LIN {X 0,Y 488.788,Z 369.847,A -85,B 0,C 180,E1 23776.764,E2 23776.764} C_VEL
LIN {X 0,Y 488.831,Z 369.841,A -85,B 0,C 180,E1 23773.364,E2 23773.364} C_VEL
LIN {X 0,Y 488.776,Z 369.84,A -85,B 0,C 180,E1 23769.895,E2 23769.895} C_VEL
LIN {X 0,Y 488.771,Z 369.837,A -85,B 0,C 180,E1 23766.342,E2 23766.342} C_VEL
LIN {X 0,Y 488.82,Z 369.843,A -85,B 0,C 180,E1 23762.931,E2 23762.931} C_VEL
LIN {X 0,Y 488.772,Z 369.849,A -85,B 0,C 180,E1 23759.531,E2 23759.531} C_VEL
LIN {X 0,Y 488.762,Z 369.849,A -85,B 0,C 180,E1 23756.012,E2 23756.012} C_VEL
LIN {X 0,Y 488.816,Z 369.838,A -85,B 0,C 180,E1 23752.596,E2 23752.596} C_VEL
LIN {X 0,Y 488.767,Z 369.845,A -85,B 0,C 180,E1 23749.152,E2 23749.152} C_VEL
LIN {X 0,Y 488.75,Z 369.847,A -85,B 0,C 180,E1 23745.669,E2 23745.669} C_VEL
LIN {X 0,Y 488.801,Z 369.846,A -85,B 0,C 180,E1 23742.255,E2 23742.255} C_VEL
LIN {X 0,Y 488.77,Z 369.853,A -85,B 0,C 180,E1 23738.772,E2 23738.772} C_VEL
LIN {X 0,Y 488.748,Z 369.822,A -85,B 0,C 180,E1 23735.262,E2 23735.262} C_VEL
LIN {X 0,Y 488.792,Z 369.844,A -85,B 0,C 180,E1 23731.802,E2 23731.802} C_VEL
LIN {X 0,Y 488.773,Z 369.83,A -85,B 0,C 180,E1 23728.535,E2 23728.535} C_VEL
LIN {X 0,Y 488.76,Z 369.829,A -85,B 0,C 180,E1 23725.055,E2 23725.055} C_VEL
LIN {X 0,Y 488.805,Z 369.844,A -85,B 0,C 180,E1 23721.55,E2 23721.55} C_VEL
LIN {X 0,Y 488.797,Z 369.846,A -85,B 0,C 180,E1 23718.117,E2 23718.117} C_VEL
LIN {X 0,Y 488.832,Z 370.155,A -85,B 0,C 180,E1 23717.192,E2 23717.192} C_VEL
LIN {X 0,Y 490.288,Z 373.622,A -85,B 0,C 180,E1 23716.717,E2 23716.717} C_VEL
LIN {X 0,Y 496.839,Z 386.984,A -85,B 0,C 180,E1 23715.06,E2 23715.06} C_VEL
LIN {X 0,Y 507.598,Z 410.407,A -85,B 0,C 180,E1 23712.424,E2 23712.424} C_VEL
LIN {X 0,Y 505.734,Z 452.561,A -85,B 0,C 180,E1 23709.796,E2 23709.796} C_VEL
LIN {X 0,Y 508.868,Z 476.154,A -85,B 0,C 180,E1 23709.124,E2 23709.124} C_VEL
LIN {X 0,Y 505.724,Z 690.25,A -85,B 0,C 180,E1 23705.753,E2 23705.753} C_VEL
LIN {X 0,Y 504.658,Z 761.758,A -85,B 0,C 180,E1 23704.625,E2 23704.625} C_VEL
LIN {X 0,Y 503.792,Z 783.614,A -85,B 0,C 180,E1 23704.081,E2 23704.081} C_VEL
LIN {X 0,Y 502.692,Z 805.814,A -85,B 0,C 180,E1 23703.323,E2 23703.323} C_VEL
LIN {X 0,Y 501.534,Z 826.289,A -85,B 0,C 180,E1 23702.427,E2 23702.427} C_VEL
LIN {X 0,Y 500.044,Z 845.014,A -85,B 0,C 180,E1 23701.373,E2 23701.373} C_VEL
LIN {X 0,Y 498.307,Z 865.526,A -85,B 0,C 180,E1 23699.972,E2 23699.972} C_VEL
LIN {X 0,Y 496.641,Z 883.778,A -85,B 0,C 180,E1 23698.496,E2 23698.496} C_VEL
LIN {X 0,Y 494.933,Z 901.869,A -85,B 0,C 180,E1 23696.758,E2 23696.758} C_VEL
LIN {X 0,Y 493.326,Z 918.685,A -85,B 0,C 180,E1 23694.867,E2 23694.867} C_VEL
LIN {X 0,Y 491.919,Z 934.189,A -85,B 0,C 180,E1 23692.842,E2 23692.842} C_VEL
LIN {X 0,Y 490.709,Z 948.64,A -85,B 0,C 180,E1 23690.639,E2 23690.639} C_VEL
LIN {X 0,Y 489.722,Z 961.46,A -85,B 0,C 180,E1 23688.324,E2 23688.324} C_VEL
LIN {X 0,Y 488.984,Z 972.816,A -85,B 0,C 180,E1 23685.901,E2 23685.901} C_VEL
LIN {X 0,Y 488.492,Z 982.262,A -85,B 0,C 180,E1 23683.493,E2 23683.493} C_VEL
LIN {X 0,Y 488.185,Z 989.884,A -85,B 0,C 180,E1 23681.099,E2 23681.099} C_VEL
LIN {X 0,Y 488.014,Z 996.146,A -85,B 0,C 180,E1 23678.601,E2 23678.601} C_VEL
LIN {X 0,Y 487.941,Z 1000.823,A -85,B 0,C 180,E1 23676.117,E2 23676.117} C_VEL
LIN {X 0,Y 487.912,Z 1003.79,A -85,B 0,C 180,E1 23673.639,E2 23673.639} C_VEL
LIN {X 0,Y 487.908,Z 1005.304,A -85,B 0,C 180,E1 23671.057,E2 23671.057} C_VEL
LIN {X 0,Y 487.907,Z 1005.259,A -85,B 0,C 180,E1 23668.709,E2 23668.709} C_VEL
LIN {X 0,Y 487.911,Z 1003.672,A -85,B 0,C 180,E1 23666.241,E2 23666.241} C_VEL
LIN {X 0,Y 487.944,Z 1000.634,A -85,B 0,C 180,E1 23663.766,E2 23663.766} C_VEL
LIN {X 0,Y 488.016,Z 995.893,A -85,B 0,C 180,E1 23661.281,E2 23661.281} C_VEL
LIN {X 0,Y 488.205,Z 989.179,A -85,B 0,C 180,E1 23658.663,E2 23658.663} C_VEL
LIN {X 0,Y 488.532,Z 981.433,A -85,B 0,C 180,E1 23656.268,E2 23656.268} C_VEL
LIN {X 0,Y 489.043,Z 971.79,A -85,B 0,C 180,E1 23653.858,E2 23653.858} C_VEL
LIN {X 0,Y 489.806,Z 960.195,A -85,B 0,C 180,E1 23651.433,E2 23651.433} C_VEL
LIN {X 0,Y 490.765,Z 947.879,A -85,B 0,C 180,E1 23649.24,E2 23649.24} C_VEL
LIN {X 0,Y 491.917,Z 934.195,A -85,B 0,C 180,E1 23647.159,E2 23647.159} C_VEL
LIN {X 0,Y 493.326,Z 918.693,A -85,B 0,C 180,E1 23645.133,E2 23645.133} C_VEL
LIN {X 0,Y 494.944,Z 901.728,A -85,B 0,C 180,E1 23643.228,E2 23643.228} C_VEL
LIN {X 0,Y 496.642,Z 883.789,A -85,B 0,C 180,E1 23641.505,E2 23641.505} C_VEL
LIN {X 0,Y 498.307,Z 865.542,A -85,B 0,C 180,E1 23640.029,E2 23640.029} C_VEL
LIN {X 0,Y 500.043,Z 845.02,A -85,B 0,C 180,E1 23638.627,E2 23638.627} C_VEL
LIN {X 0,Y 501.533,Z 826.306,A -85,B 0,C 180,E1 23637.573,E2 23637.573} C_VEL
LIN {X 0,Y 502.7,Z 805.692,A -85,B 0,C 180,E1 23636.671,E2 23636.671} C_VEL
LIN {X 0,Y 503.838,Z 782.562,A -85,B 0,C 180,E1 23635.889,E2 23635.889} C_VEL
LIN {X 0,Y 504.681,Z 760.801,A -85,B 0,C 180,E1 23635.356,E2 23635.356} C_VEL
LIN {X 0,Y 507.814,Z 542.394,A -85,B 0,C 180,E1 23631.935,E2 23631.935} C_VEL
LIN {X 0,Y 508.709,Z 473.556,A -85,B 0,C 180,E1 23630.818,E2 23630.818} C_VEL
LIN {X 0,Y 505.659,Z 451.562,A -85,B 0,C 180,E1 23630.164,E2 23630.164} C_VEL
LIN {X 0,Y 507.487,Z 410.144,A -85,B 0,C 180,E1 23627.548,E2 23627.548} C_VEL
LIN {X 0,Y 496.402,Z 386,A -85,B 0,C 180,E1 23624.827,E2 23624.827} C_VEL
LIN {X 0,Y 490.187,Z 373.48,A -85,B 0,C 180,E1 23623.263,E2 23623.263} C_VEL
LIN {X 0,Y 488.827,Z 370.128,A -85,B 0,C 180,E1 23622.809,E2 23622.809} C_VEL
LIN {X 0,Y 488.765,Z 369.836,A -85,B 0,C 180,E1 23621.35,E2 23621.35} C_VEL
LIN {X 0,Y 488.818,Z 369.85,A -85,B 0,C 180,E1 23618.001,E2 23618.001} C_VEL
LIN {X 0,Y 488.785,Z 369.834,A -85,B 0,C 180,E1 23614.484,E2 23614.484} C_VEL
LIN {X 0,Y 488.756,Z 369.825,A -85,B 0,C 180,E1 23611.012,E2 23611.012} C_VEL
LIN {X 0,Y 488.805,Z 369.85,A -85,B 0,C 180,E1 23607.667,E2 23607.667} C_VEL
LIN {X 0,Y 488.766,Z 369.816,A -85,B 0,C 180,E1 23604.279,E2 23604.279} C_VEL
LIN {X 0,Y 488.752,Z 369.852,A -85,B 0,C 180,E1 23600.804,E2 23600.804} C_VEL
LIN {X 0,Y 488.797,Z 369.851,A -85,B 0,C 180,E1 23597.376,E2 23597.376} C_VEL
LIN {X 0,Y 488.766,Z 369.847,A -85,B 0,C 180,E1 23593.968,E2 23593.968} C_VEL
LIN {X 0,Y 488.75,Z 369.847,A -85,B 0,C 180,E1 23590.49,E2 23590.49} C_VEL
LIN {X 0,Y 488.798,Z 369.839,A -85,B 0,C 180,E1 23587.05,E2 23587.05} C_VEL
LIN {X 0,Y 488.778,Z 369.848,A -85,B 0,C 180,E1 23583.636,E2 23583.636} C_VEL
LIN {X 0,Y 488.758,Z 369.85,A -85,B 0,C 180,E1 23580.117,E2 23580.117} C_VEL
LIN {X 0,Y 488.803,Z 369.848,A -85,B 0,C 180,E1 23576.716,E2 23576.716} C_VEL
LIN {X 0,Y 488.789,Z 369.837,A -85,B 0,C 180,E1 23573.304,E2 23573.304} C_VEL
LIN {X 0,Y 488.766,Z 369.839,A -85,B 0,C 180,E1 23569.867,E2 23569.867} C_VEL
LIN {X 0,Y 488.809,Z 369.841,A -85,B 0,C 180,E1 23566.394,E2 23566.394} C_VEL
LIN {X 0,Y 488.801,Z 369.849,A -85,B 0,C 180,E1 23562.991,E2 23562.991} C_VEL
LIN {X 0,Y 488.777,Z 369.846,A -85,B 0,C 180,E1 23559.521,E2 23559.521} C_VEL
LIN {X 0,Y 488.815,Z 369.843,A -85,B 0,C 180,E1 23556.096,E2 23556.096} C_VEL
LIN {X 0,Y 488.819,Z 369.838,A -85,B 0,C 180,E1 23552.577,E2 23552.577} C_VEL
LIN {X 0,Y 488.783,Z 369.839,A -85,B 0,C 180,E1 23549.106,E2 23549.106} C_VEL
LIN {X 0,Y 488.809,Z 369.841,A -85,B 0,C 180,E1 23545.628,E2 23545.628} C_VEL
LIN {X 0,Y 488.829,Z 369.815,A -85,B 0,C 180,E1 23542.134,E2 23542.134} C_VEL
LIN {X 0,Y 488.796,Z 369.848,A -85,B 0,C 180,E1 23538.645,E2 23538.645} C_VEL
LIN {X 0,Y 488.797,Z 369.824,A -85,B 0,C 180,E1 23535.047,E2 23535.047} C_VEL
LIN {X 0,Y 488.833,Z 369.816,A -85,B 0,C 180,E1 23531.501,E2 23531.501} C_VEL
LIN {X 0,Y 488.829,Z 369.836,A -85,B 0,C 180,E1 23527.858,E2 23527.858} C_VEL
LIN {X 0,Y 489.015,Z 370.806,A -85,B 0,C 180,E1 23527.599,E2 23527.599} C_VEL
LIN {X 0,Y 494.904,Z 385.117,A -85,B 0,C 180,E1 23525.426,E2 23525.426} C_VEL
LIN {X 0,Y 496.471,Z 389.129,A -85,B 0,C 180,E1 23525.033,E2 23525.033} C_VEL
LIN {X 0,Y 498.27,Z 395.004,A -85,B 0,C 180,E1 23524.736,E2 23524.736} C_VEL
LIN {X 0,Y 499.36,Z 402.645,A -85,B 0,C 180,E1 23524.515,E2 23524.515} C_VEL
LIN {X 0,Y 499.244,Z 418.921,A -85,B 0,C 180,E1 23524.239,E2 23524.239} C_VEL
LIN {X 0,Y 495.859,Z 645.556,A -85,B 0,C 180,E1 23520.716,E2 23520.716} C_VEL
LIN {X 0,Y 495.214,Z 666.185,A -85,B 0,C 180,E1 23520.218,E2 23520.218} C_VEL
LIN {X 0,Y 494.31,Z 684.909,A -85,B 0,C 180,E1 23519.567,E2 23519.567} C_VEL
LIN {X 0,Y 493.108,Z 703.249,A -85,B 0,C 180,E1 23518.718,E2 23518.718} C_VEL
LIN {X 0,Y 491.661,Z 720.942,A -85,B 0,C 180,E1 23517.686,E2 23517.686} C_VEL
LIN {X 0,Y 489.933,Z 739.495,A -85,B 0,C 180,E1 23516.355,E2 23516.355} C_VEL
LIN {X 0,Y 488.265,Z 755.721,A -85,B 0,C 180,E1 23514.948,E2 23514.948} C_VEL
LIN {X 0,Y 486.607,Z 771.11,A -85,B 0,C 180,E1 23513.361,E2 23513.361} C_VEL
LIN {X 0,Y 484.95,Z 785.984,A -85,B 0,C 180,E1 23511.528,E2 23511.528} C_VEL
LIN {X 0,Y 483.466,Z 799.353,A -85,B 0,C 180,E1 23509.572,E2 23509.572} C_VEL
LIN {X 0,Y 482.254,Z 811.31,A -85,B 0,C 180,E1 23507.493,E2 23507.493} C_VEL
LIN {X 0,Y 481.219,Z 822.432,A -85,B 0,C 180,E1 23505.175,E2 23505.175} C_VEL
LIN {X 0,Y 480.437,Z 834.341,A -85,B 0,C 180,E1 23502.132,E2 23502.132} C_VEL
LIN {X 0,Y 480.148,Z 841.698,A -85,B 0,C 180,E1 23499.83,E2 23499.83} C_VEL
LIN {X 0,Y 479.982,Z 847.651,A -85,B 0,C 180,E1 23497.419,E2 23497.419} C_VEL
LIN {X 0,Y 479.922,Z 851.89,A -85,B 0,C 180,E1 23495.019,E2 23495.019} C_VEL
LIN {X 0,Y 479.912,Z 854.507,A -85,B 0,C 180,E1 23492.626,E2 23492.626} C_VEL
LIN {X 0,Y 479.908,Z 855.453,A -85,B 0,C 180,E1 23490.238,E2 23490.238} C_VEL
LIN {X 0,Y 479.912,Z 854.828,A -85,B 0,C 180,E1 23487.851,E2 23487.851} C_VEL
LIN {X 0,Y 479.923,Z 852.487,A -85,B 0,C 180,E1 23485.34,E2 23485.34} C_VEL
LIN {X 0,Y 479.972,Z 848.604,A -85,B 0,C 180,E1 23482.94,E2 23482.94} C_VEL
LIN {X 0,Y 480.107,Z 842.998,A -85,B 0,C 180,E1 23480.531,E2 23480.531} C_VEL
LIN {X 0,Y 480.37,Z 835.903,A -85,B 0,C 180,E1 23478.231,E2 23478.231} C_VEL
LIN {X 0,Y 481.095,Z 824.054,A -85,B 0,C 180,E1 23475.108,E2 23475.108} C_VEL
LIN {X 0,Y 482.034,Z 813.717,A -85,B 0,C 180,E1 23472.871,E2 23472.871} C_VEL
LIN {X 0,Y 483.282,Z 801.241,A -85,B 0,C 180,E1 23470.634,E2 23470.634} C_VEL
LIN {X 0,Y 484.778,Z 787.534,A -85,B 0,C 180,E1 23468.59,E2 23468.59} C_VEL
LIN {X 0,Y 486.38,Z 772.874,A -85,B 0,C 180,E1 23466.755,E2 23466.755} C_VEL
LIN {X 0,Y 488.076,Z 757.496,A -85,B 0,C 180,E1 23465.136,E2 23465.136} C_VEL
LIN {X 0,Y 489.807,Z 740.762,A -85,B 0,C 180,E1 23463.656,E2 23463.656} C_VEL
LIN {X 0,Y 491.484,Z 723.176,A -85,B 0,C 180,E1 23462.368,E2 23462.368} C_VEL
LIN {X 0,Y 492.997,Z 704.892,A -85,B 0,C 180,E1 23461.274,E2 23461.274} C_VEL
LIN {X 0,Y 494.242,Z 686.026,A -85,B 0,C 180,E1 23460.391,E2 23460.391} C_VEL
LIN {X 0,Y 495.212,Z 666.341,A -85,B 0,C 180,E1 23459.696,E2 23459.696} C_VEL
LIN {X 0,Y 495.868,Z 645.599,A -85,B 0,C 180,E1 23459.193,E2 23459.193} C_VEL
LIN {X 0,Y 499.057,Z 431.182,A -85,B 0,C 180,E1 23455.86,E2 23455.86} C_VEL
LIN {X 0,Y 499.3,Z 407.126,A -85,B 0,C 180,E1 23455.472,E2 23455.472} C_VEL
LIN {X 0,Y 489.488,Z 390.831,A -85,B 0,C 180,E1 23454.288,E2 23454.288} C_VEL
LIN {X 0,Y 487.873,Z 387.972,A -85,B 0,C 180,E1 23454.05,E2 23454.05} C_VEL
LIN {X 0,Y 481.849,Z 373.753,A -85,B 0,C 180,E1 23451.855,E2 23451.855} C_VEL
LIN {X 0,Y 480.889,Z 371.018,A -85,B 0,C 180,E1 23451.375,E2 23451.375} C_VEL
LIN {X 0,Y 480.884,Z 370.81,A -85,B 0,C 180,E1 23447.926,E2 23447.926} C_VEL
LIN {X 0,Y 480.889,Z 370.803,A -85,B 0,C 180,E1 23444.316,E2 23444.316} C_VEL
LIN {X 0,Y 480.864,Z 370.834,A -85,B 0,C 180,E1 23440.761,E2 23440.761} C_VEL
LIN {X 0,Y 480.855,Z 370.824,A -85,B 0,C 180,E1 23437.086,E2 23437.086} C_VEL
LIN {X 0,Y 480.883,Z 370.829,A -85,B 0,C 180,E1 23433.521,E2 23433.521} C_VEL
LIN {X 0,Y 480.899,Z 370.824,A -85,B 0,C 180,E1 23429.897,E2 23429.897} C_VEL
LIN {X 0,Y 480.853,Z 370.829,A -85,B 0,C 180,E1 23426.348,E2 23426.348} C_VEL
LIN {X 0,Y 480.847,Z 370.83,A -85,B 0,C 180,E1 23422.754,E2 23422.754} C_VEL
LIN {X 0,Y 480.887,Z 370.824,A -85,B 0,C 180,E1 23419.289,E2 23419.289} C_VEL
LIN {X 0,Y 480.868,Z 370.833,A -85,B 0,C 180,E1 23415.716,E2 23415.716} C_VEL
LIN {X 0,Y 480.833,Z 370.837,A -85,B 0,C 180,E1 23412.246,E2 23412.246} C_VEL
LIN {X 0,Y 480.856,Z 370.839,A -85,B 0,C 180,E1 23408.731,E2 23408.731} C_VEL
LIN {X 0,Y 480.875,Z 370.824,A -85,B 0,C 180,E1 23405.249,E2 23405.249} C_VEL
LIN {X 0,Y 480.827,Z 370.827,A -85,B 0,C 180,E1 23401.788,E2 23401.788} C_VEL
LIN {X 0,Y 480.831,Z 370.832,A -85,B 0,C 180,E1 23398.213,E2 23398.213} C_VEL
LIN {X 0,Y 480.879,Z 370.837,A -85,B 0,C 180,E1 23394.751,E2 23394.751} C_VEL
LIN {X 0,Y 480.821,Z 370.837,A -85,B 0,C 180,E1 23391.389,E2 23391.389} C_VEL
LIN {X 0,Y 480.815,Z 370.839,A -85,B 0,C 180,E1 23387.754,E2 23387.754} C_VEL
LIN {X 0,Y 480.859,Z 370.831,A -85,B 0,C 180,E1 23384.288,E2 23384.288} C_VEL
LIN {X 0,Y 480.83,Z 370.831,A -85,B 0,C 180,E1 23380.819,E2 23380.819} C_VEL
LIN {X 0,Y 480.811,Z 370.828,A -85,B 0,C 180,E1 23377.374,E2 23377.374} C_VEL
LIN {X 0,Y 480.856,Z 370.825,A -85,B 0,C 180,E1 23373.921,E2 23373.921} C_VEL
LIN {X 0,Y 480.833,Z 370.816,A -85,B 0,C 180,E1 23370.598,E2 23370.598} C_VEL
LIN {X 0,Y 480.823,Z 370.842,A -85,B 0,C 180,E1 23367.13,E2 23367.13} C_VEL
LIN {X 0,Y 480.864,Z 370.809,A -85,B 0,C 180,E1 23363.659,E2 23363.659} C_VEL
LIN {X 0,Y 480.842,Z 370.812,A -85,B 0,C 180,E1 23360.291,E2 23360.291} C_VEL
LIN {X 0,Y 480.881,Z 370.964,A -85,B 0,C 180,E1 23358.051,E2 23358.051} C_VEL
LIN {X 0,Y 481.309,Z 372.589,A -85,B 0,C 180,E1 23357.777,E2 23357.777} C_VEL
LIN {X 0,Y 488.746,Z 387.377,A -85,B 0,C 180,E1 23355.847,E2 23355.847} C_VEL
LIN {X 0,Y 498.284,Z 408.17,A -85,B 0,C 180,E1 23353.416,E2 23353.416} C_VEL
LIN {X 0,Y 500.866,Z 414.181,A -85,B 0,C 180,E1 23352.763,E2 23352.763} C_VEL
LIN {X 0,Y 499.003,Z 451.774,A -85,B 0,C 180,E1 23350.384,E2 23350.384} C_VEL
LIN {X 0,Y 502.359,Z 477.415,A -85,B 0,C 180,E1 23349.638,E2 23349.638} C_VEL
LIN {X 0,Y 498.808,Z 694.303,A -85,B 0,C 180,E1 23346.163,E2 23346.163} C_VEL
LIN {X 0,Y 497.703,Z 760.723,A -85,B 0,C 180,E1 23345.096,E2 23345.096} C_VEL
LIN {X 0,Y 496.779,Z 782.356,A -85,B 0,C 180,E1 23344.552,E2 23344.552} C_VEL
LIN {X 0,Y 495.548,Z 804.985,A -85,B 0,C 180,E1 23343.77,E2 23343.77} C_VEL
LIN {X 0,Y 494.251,Z 826.148,A -85,B 0,C 180,E1 23342.827,E2 23342.827} C_VEL
LIN {X 0,Y 492.717,Z 846.558,A -85,B 0,C 180,E1 23341.704,E2 23341.704} C_VEL
LIN {X 0,Y 491.223,Z 865.433,A -85,B 0,C 180,E1 23340.45,E2 23340.45} C_VEL
LIN {X 0,Y 489.581,Z 882.526,A -85,B 0,C 180,E1 23339.063,E2 23339.063} C_VEL
LIN {X 0,Y 487.818,Z 899.472,A -85,B 0,C 180,E1 23337.44,E2 23337.44} C_VEL
LIN {X 0,Y 486.066,Z 916.658,A -85,B 0,C 180,E1 23335.526,E2 23335.526} C_VEL
LIN {X 0,Y 484.509,Z 932.49,A -85,B 0,C 180,E1 23333.469,E2 23333.469} C_VEL
LIN {X 0,Y 483.124,Z 947.102,A -85,B 0,C 180,E1 23331.232,E2 23331.232} C_VEL
LIN {X 0,Y 482.029,Z 959.88,A -85,B 0,C 180,E1 23328.939,E2 23328.939} C_VEL
LIN {X 0,Y 481.194,Z 971.27,A -85,B 0,C 180,E1 23326.538,E2 23326.538} C_VEL
LIN {X 0,Y 480.617,Z 980.974,A -85,B 0,C 180,E1 23324.086,E2 23324.086} C_VEL
LIN {X 0,Y 480.251,Z 988.824,A -85,B 0,C 180,E1 23321.65,E2 23321.65} C_VEL
LIN {X 0,Y 480.046,Z 995.384,A -85,B 0,C 180,E1 23319.107,E2 23319.107} C_VEL
LIN {X 0,Y 479.956,Z 1000.019,A -85,B 0,C 180,E1 23316.699,E2 23316.699} C_VEL
LIN {X 0,Y 479.915,Z 1003.446,A -85,B 0,C 180,E1 23314.062,E2 23314.062} C_VEL
LIN {X 0,Y 479.9,Z 1005.209,A -85,B 0,C 180,E1 23311.552,E2 23311.552} C_VEL
LIN {X 0,Y 479.903,Z 1005.326,A -85,B 0,C 180,E1 23309.045,E2 23309.045} C_VEL
LIN {X 0,Y 479.912,Z 1003.899,A -85,B 0,C 180,E1 23306.417,E2 23306.417} C_VEL
LIN {X 0,Y 479.943,Z 1000.98,A -85,B 0,C 180,E1 23303.902,E2 23303.902} C_VEL
LIN {X 0,Y 480.02,Z 996.401,A -85,B 0,C 180,E1 23301.376,E2 23301.376} C_VEL
LIN {X 0,Y 480.203,Z 990.238,A -85,B 0,C 180,E1 23298.836,E2 23298.836} C_VEL
LIN {X 0,Y 480.548,Z 982.419,A -85,B 0,C 180,E1 23296.328,E2 23296.328} C_VEL
LIN {X 0,Y 481.099,Z 972.817,A -85,B 0,C 180,E1 23293.832,E2 23293.832} C_VEL
LIN {X 0,Y 481.911,Z 961.463,A -85,B 0,C 180,E1 23291.369,E2 23291.369} C_VEL
LIN {X 0,Y 482.93,Z 949.363,A -85,B 0,C 180,E1 23289.141,E2 23289.141} C_VEL
LIN {X 0,Y 484.149,Z 935.883,A -85,B 0,C 180,E1 23287.028,E2 23287.028} C_VEL
LIN {X 0,Y 485.751,Z 919.705,A -85,B 0,C 180,E1 23284.849,E2 23284.849} C_VEL
LIN {X 0,Y 487.435,Z 903.548,A -85,B 0,C 180,E1 23282.98,E2 23282.98} C_VEL
LIN {X 0,Y 489.185,Z 886.121,A -85,B 0,C 180,E1 23281.263,E2 23281.263} C_VEL
LIN {X 0,Y 491,Z 867.941,A -85,B 0,C 180,E1 23279.739,E2 23279.739} C_VEL
LIN {X 0,Y 492.26,Z 852.622,A -85,B 0,C 180,E1 23278.673,E2 23278.673} C_VEL
LIN {X 0,Y 493.82,Z 831.791,A -85,B 0,C 180,E1 23277.465,E2 23277.465} C_VEL
LIN {X 0,Y 495.244,Z 810.72,A -85,B 0,C 180,E1 23276.461,E2 23276.461} C_VEL
LIN {X 0,Y 496.444,Z 788.83,A -85,B 0,C 180,E1 23275.645,E2 23275.645} C_VEL
LIN {X 0,Y 497.445,Z 767.04,A -85,B 0,C 180,E1 23275.048,E2 23275.048} C_VEL
LIN {X 0,Y 498.113,Z 742.947,A -85,B 0,C 180,E1 23274.597,E2 23274.597} C_VEL
LIN {X 0,Y 501.442,Z 527.679,A -85,B 0,C 180,E1 23271.181,E2 23271.181} C_VEL
LIN {X 0,Y 502.21,Z 474.909,A -85,B 0,C 180,E1 23270.305,E2 23270.305} C_VEL
LIN {X 0,Y 498.951,Z 450.509,A -85,B 0,C 180,E1 23269.558,E2 23269.558} C_VEL
LIN {X 0,Y 500.826,Z 413.756,A -85,B 0,C 180,E1 23267.204,E2 23267.204} C_VEL
LIN {X 0,Y 490.266,Z 390.634,A -85,B 0,C 180,E1 23264.552,E2 23264.552} C_VEL
LIN {X 0,Y 482.4,Z 374.624,A -85,B 0,C 180,E1 23262.507,E2 23262.507} C_VEL
LIN {X 0,Y 480.92,Z 371.178,A -85,B 0,C 180,E1 23262.025,E2 23262.025} C_VEL
LIN {X 0,Y 480.826,Z 370.823,A -85,B 0,C 180,E1 23261.357,E2 23261.357} C_VEL
LIN {X 0,Y 480.877,Z 370.839,A -85,B 0,C 180,E1 23257.985,E2 23257.985} C_VEL
LIN {X 0,Y 480.857,Z 370.822,A -85,B 0,C 180,E1 23254.371,E2 23254.371} C_VEL
LIN {X 0,Y 480.817,Z 370.81,A -85,B 0,C 180,E1 23250.906,E2 23250.906} C_VEL
LIN {X 0,Y 480.841,Z 370.84,A -85,B 0,C 180,E1 23247.401,E2 23247.401} C_VEL
LIN {X 0,Y 480.862,Z 370.799,A -85,B 0,C 180,E1 23243.92,E2 23243.92} C_VEL
LIN {X 0,Y 480.812,Z 370.841,A -85,B 0,C 180,E1 23240.575,E2 23240.575} C_VEL
LIN {X 0,Y 480.821,Z 370.84,A -85,B 0,C 180,E1 23236.97,E2 23236.97} C_VEL
LIN {X 0,Y 480.874,Z 370.837,A -85,B 0,C 180,E1 23233.466,E2 23233.466} C_VEL
LIN {X 0,Y 480.825,Z 370.836,A -85,B 0,C 180,E1 23229.938,E2 23229.938} C_VEL
LIN {X 0,Y 480.815,Z 370.835,A -85,B 0,C 180,E1 23226.447,E2 23226.447} C_VEL
LIN {X 0,Y 480.866,Z 370.826,A -85,B 0,C 180,E1 23222.979,E2 23222.979} C_VEL
LIN {X 0,Y 480.842,Z 370.838,A -85,B 0,C 180,E1 23219.523,E2 23219.523} C_VEL
LIN {X 0,Y 480.825,Z 370.837,A -85,B 0,C 180,E1 23216.065,E2 23216.065} C_VEL
LIN {X 0,Y 480.867,Z 370.835,A -85,B 0,C 180,E1 23212.593,E2 23212.593} C_VEL
LIN {X 0,Y 480.862,Z 370.825,A -85,B 0,C 180,E1 23209.093,E2 23209.093} C_VEL
LIN {X 0,Y 480.83,Z 370.831,A -85,B 0,C 180,E1 23205.673,E2 23205.673} C_VEL
LIN {X 0,Y 480.866,Z 370.831,A -85,B 0,C 180,E1 23202.202,E2 23202.202} C_VEL
LIN {X 0,Y 480.887,Z 370.836,A -85,B 0,C 180,E1 23198.651,E2 23198.651} C_VEL
LIN {X 0,Y 480.843,Z 370.836,A -85,B 0,C 180,E1 23195.163,E2 23195.163} C_VEL
LIN {X 0,Y 480.852,Z 370.835,A -85,B 0,C 180,E1 23191.564,E2 23191.564} C_VEL
LIN {X 0,Y 480.897,Z 370.833,A -85,B 0,C 180,E1 23188.122,E2 23188.122} C_VEL
LIN {X 0,Y 480.868,Z 370.836,A -85,B 0,C 180,E1 23184.541,E2 23184.541} C_VEL
LIN {X 0,Y 480.847,Z 370.801,A -85,B 0,C 180,E1 23180.946,E2 23180.946} C_VEL
LIN {X 0,Y 480.874,Z 370.828,A -85,B 0,C 180,E1 23177.39,E2 23177.39} C_VEL
LIN {X 0,Y 480.895,Z 370.83,A -85,B 0,C 180,E1 23173.811,E2 23173.811} C_VEL
LIN {X 0,Y 480.866,Z 370.813,A -85,B 0,C 180,E1 23170.262,E2 23170.262} C_VEL
LIN {X 0,Y 480.892,Z 371.07,A -85,B 0,C 180,E1 23168.509,E2 23168.509} C_VEL
LIN {X 0,Y 486.764,Z 385.17,A -85,B 0,C 180,E1 23166.264,E2 23166.264} C_VEL
LIN {X 0,Y 488.473,Z 389.111,A -85,B 0,C 180,E1 23165.747,E2 23165.747} C_VEL
LIN {X 0,Y 499.31,Z 407.175,A -85,B 0,C 180,E1 23164.434,E2 23164.434} C_VEL
LIN {X 0,Y 499.244,Z 418.921,A -85,B 0,C 180,E1 23164.239,E2 23164.239} C_VEL
LIN {X 0,Y 498.378,Z 426.618,A -85,B 0,C 180,E1 23164.185,E2 23164.185} C_VEL
LIN {X 0,Y 493.068,Z 447.174,A -85,B 0,C 180,E1 23164.308,E2 23164.308} C_VEL
LIN {X 0,Y 492.343,Z 453.787,A -85,B 0,C 180,E1 23164.26,E2 23164.26} C_VEL
LIN {X 0,Y 489.336,Z 650.297,A -85,B 0,C 180,E1 23161.184,E2 23161.184} C_VEL
LIN {X 0,Y 488.616,Z 670.204,A -85,B 0,C 180,E1 23160.663,E2 23160.663} C_VEL
LIN {X 0,Y 487.592,Z 689.333,A -85,B 0,C 180,E1 23159.951,E2 23159.951} C_VEL
LIN {X 0,Y 486.282,Z 707.632,A -85,B 0,C 180,E1 23159.066,E2 23159.066} C_VEL
LIN {X 0,Y 484.66,Z 726.308,A -85,B 0,C 180,E1 23157.921,E2 23157.921} C_VEL
LIN {X 0,Y 482.882,Z 743.342,A -85,B 0,C 180,E1 23156.63,E2 23156.63} C_VEL
LIN {X 0,Y 481.042,Z 759.594,A -85,B 0,C 180,E1 23155.151,E2 23155.151} C_VEL
LIN {X 0,Y 479.062,Z 776.072,A -85,B 0,C 180,E1 23153.36,E2 23153.36} C_VEL
LIN {X 0,Y 477.354,Z 790.398,A -85,B 0,C 180,E1 23151.5,E2 23151.5} C_VEL
LIN {X 0,Y 475.822,Z 803.326,A -85,B 0,C 180,E1 23149.516,E2 23149.516} C_VEL
LIN {X 0,Y 474.494,Z 815.492,A -85,B 0,C 180,E1 23147.282,E2 23147.282} C_VEL
LIN {X 0,Y 473.425,Z 826.079,A -85,B 0,C 180,E1 23144.929,E2 23144.929} C_VEL
LIN {X 0,Y 472.717,Z 834.698,A -85,B 0,C 180,E1 23142.582,E2 23142.582} C_VEL
LIN {X 0,Y 472.227,Z 842.036,A -85,B 0,C 180,E1 23140.081,E2 23140.081} C_VEL
LIN {X 0,Y 471.994,Z 847.767,A -85,B 0,C 180,E1 23137.519,E2 23137.519} C_VEL
LIN {X 0,Y 471.925,Z 852.209,A -85,B 0,C 180,E1 23134.861,E2 23134.861} C_VEL
LIN {X 0,Y 471.91,Z 854.643,A -85,B 0,C 180,E1 23132.428,E2 23132.428} C_VEL
LIN {X 0,Y 471.914,Z 855.497,A -85,B 0,C 180,E1 23130,E2 23130} C_VEL
LIN {X 0,Y 471.906,Z 854.691,A -85,B 0,C 180,E1 23127.571,E2 23127.571} C_VEL
LIN {X 0,Y 471.925,Z 852.325,A -85,B 0,C 180,E1 23125.139,E2 23125.139} C_VEL
LIN {X 0,Y 471.985,Z 848.136,A -85,B 0,C 180,E1 23122.576,E2 23122.576} C_VEL
LIN {X 0,Y 472.209,Z 842.497,A -85,B 0,C 180,E1 23120.002,E2 23120.002} C_VEL
LIN {X 0,Y 472.662,Z 835.424,A -85,B 0,C 180,E1 23117.54,E2 23117.54} C_VEL
LIN {X 0,Y 473.395,Z 826.454,A -85,B 0,C 180,E1 23115.069,E2 23115.069} C_VEL
LIN {X 0,Y 474.463,Z 815.719,A -85,B 0,C 180,E1 23112.675,E2 23112.675} C_VEL
LIN {X 0,Y 475.757,Z 803.827,A -85,B 0,C 180,E1 23110.48,E2 23110.48} C_VEL
LIN {X 0,Y 477.327,Z 790.636,A -85,B 0,C 180,E1 23108.443,E2 23108.443} C_VEL
LIN {X 0,Y 479.043,Z 776.263,A -85,B 0,C 180,E1 23106.573,E2 23106.573} C_VEL
LIN {X 0,Y 481.02,Z 759.818,A -85,B 0,C 180,E1 23104.781,E2 23104.781} C_VEL
LIN {X 0,Y 482.857,Z 743.605,A -85,B 0,C 180,E1 23103.301,E2 23103.301} C_VEL
LIN {X 0,Y 484.636,Z 726.593,A -85,B 0,C 180,E1 23102.008,E2 23102.008} C_VEL
LIN {X 0,Y 486.181,Z 708.756,A -85,B 0,C 180,E1 23100.907,E2 23100.907} C_VEL
LIN {X 0,Y 487.52,Z 690.499,A -85,B 0,C 180,E1 23100.009,E2 23100.009} C_VEL
LIN {X 0,Y 488.583,Z 671.076,A -85,B 0,C 180,E1 23099.274,E2 23099.274} C_VEL
LIN {X 0,Y 489.328,Z 651.025,A -85,B 0,C 180,E1 23098.74,E2 23098.74} C_VEL
LIN {X 0,Y 490.735,Z 559.481,A -85,B 0,C 180,E1 23097.289,E2 23097.289} C_VEL
LIN {X 0,Y 492.915,Z 410,A -85,B 0,C 180,E1 23094.944,E2 23094.944} C_VEL
LIN {X 0,Y 480.107,Z 389.093,A -85,B 0,C 180,E1 23093.327,E2 23093.327} C_VEL
LIN {X 0,Y 474.497,Z 375.687,A -85,B 0,C 180,E1 23091.23,E2 23091.23} C_VEL
LIN {X 0,Y 472.989,Z 372.055,A -85,B 0,C 180,E1 23090.581,E2 23090.581} C_VEL
LIN {X 0,Y 472.921,Z 371.817,A -85,B 0,C 180,E1 23087.192,E2 23087.192} C_VEL
LIN {X 0,Y 472.929,Z 371.796,A -85,B 0,C 180,E1 23083.523,E2 23083.523} C_VEL
LIN {X 0,Y 472.954,Z 371.794,A -85,B 0,C 180,E1 23079.885,E2 23079.885} C_VEL
LIN {X 0,Y 472.942,Z 371.82,A -85,B 0,C 180,E1 23076.296,E2 23076.296} C_VEL
LIN {X 0,Y 472.915,Z 371.825,A -85,B 0,C 180,E1 23072.713,E2 23072.713} C_VEL
LIN {X 0,Y 472.922,Z 371.827,A -85,B 0,C 180,E1 23069.096,E2 23069.096} C_VEL
LIN {X 0,Y 472.95,Z 371.821,A -85,B 0,C 180,E1 23065.494,E2 23065.494} C_VEL
LIN {X 0,Y 472.936,Z 371.818,A -85,B 0,C 180,E1 23061.871,E2 23061.871} C_VEL
LIN {X 0,Y 472.902,Z 371.82,A -85,B 0,C 180,E1 23058.335,E2 23058.335} C_VEL
LIN {X 0,Y 472.907,Z 371.817,A -85,B 0,C 180,E1 23054.698,E2 23054.698} C_VEL
LIN {X 0,Y 472.949,Z 371.815,A -85,B 0,C 180,E1 23051.216,E2 23051.216} C_VEL
LIN {X 0,Y 472.909,Z 371.825,A -85,B 0,C 180,E1 23047.655,E2 23047.655} C_VEL
LIN {X 0,Y 472.89,Z 371.827,A -85,B 0,C 180,E1 23044.123,E2 23044.123} C_VEL
LIN {X 0,Y 472.92,Z 371.821,A -85,B 0,C 180,E1 23040.606,E2 23040.606} C_VEL
LIN {X 0,Y 472.92,Z 371.815,A -85,B 0,C 180,E1 23037.092,E2 23037.092} C_VEL
LIN {X 0,Y 472.88,Z 371.823,A -85,B 0,C 180,E1 23033.566,E2 23033.566} C_VEL
LIN {X 0,Y 472.88,Z 371.825,A -85,B 0,C 180,E1 23029.893,E2 23029.893} C_VEL
LIN {X 0,Y 472.931,Z 371.825,A -85,B 0,C 180,E1 23026.428,E2 23026.428} C_VEL
LIN {X 0,Y 472.894,Z 371.829,A -85,B 0,C 180,E1 23022.861,E2 23022.861} C_VEL
LIN {X 0,Y 472.871,Z 371.831,A -85,B 0,C 180,E1 23019.323,E2 23019.323} C_VEL
LIN {X 0,Y 472.892,Z 371.789,A -85,B 0,C 180,E1 23015.784,E2 23015.784} C_VEL
LIN {X 0,Y 472.93,Z 371.827,A -85,B 0,C 180,E1 23012.282,E2 23012.282} C_VEL
LIN {X 0,Y 472.879,Z 371.799,A -85,B 0,C 180,E1 23008.899,E2 23008.899} C_VEL
LIN {X 0,Y 472.894,Z 371.805,A -85,B 0,C 180,E1 23005.326,E2 23005.326} C_VEL
LIN {X 0,Y 472.947,Z 371.822,A -85,B 0,C 180,E1 23001.726,E2 23001.726} C_VEL
LIN {X 0,Y 472.91,Z 371.967,A -85,B 0,C 180,E1 22998.888,E2 22998.888} C_VEL
LIN {X 0,Y 473.33,Z 373.614,A -85,B 0,C 180,E1 22998.611,E2 22998.611} C_VEL
LIN {X 0,Y 475.493,Z 377.652,A -85,B 0,C 180,E1 22998.035,E2 22998.035} C_VEL
LIN {X 0,Y 483.703,Z 394.372,A -85,B 0,C 180,E1 22995.845,E2 22995.845} C_VEL
LIN {X 0,Y 492.305,Z 413.289,A -85,B 0,C 180,E1 22993.611,E2 22993.611} C_VEL
LIN {X 0,Y 494.169,Z 417.443,A -85,B 0,C 180,E1 22993.143,E2 22993.143} C_VEL
LIN {X 0,Y 492.34,Z 451.126,A -85,B 0,C 180,E1 22990.983,E2 22990.983} C_VEL
LIN {X 0,Y 495.876,Z 478.8,A -85,B 0,C 180,E1 22990.161,E2 22990.161} C_VEL
LIN {X 0,Y 491.891,Z 700.139,A -85,B 0,C 180,E1 22986.556,E2 22986.556} C_VEL
LIN {X 0,Y 490.783,Z 759.683,A -85,B 0,C 180,E1 22985.58,E2 22985.58} C_VEL
LIN {X 0,Y 489.779,Z 781.518,A -85,B 0,C 180,E1 22985.023,E2 22985.023} C_VEL
LIN {X 0,Y 488.488,Z 803.557,A -85,B 0,C 180,E1 22984.252,E2 22984.252} C_VEL
LIN {X 0,Y 487.068,Z 824.691,A -85,B 0,C 180,E1 22983.304,E2 22983.304} C_VEL
LIN {X 0,Y 485.445,Z 845.141,A -85,B 0,C 180,E1 22982.165,E2 22982.165} C_VEL
LIN {X 0,Y 483.769,Z 865.033,A -85,B 0,C 180,E1 22980.832,E2 22980.832} C_VEL
LIN {X 0,Y 482.031,Z 884.412,A -85,B 0,C 180,E1 22979.307,E2 22979.307} C_VEL
LIN {X 0,Y 480.683,Z 898.049,A -85,B 0,C 180,E1 22978.038,E2 22978.038} C_VEL
LIN {X 0,Y 478.883,Z 914.63,A -85,B 0,C 180,E1 22976.203,E2 22976.203} C_VEL
LIN {X 0,Y 477.209,Z 929.734,A -85,B 0,C 180,E1 22974.244,E2 22974.244} C_VEL
LIN {X 0,Y 475.694,Z 944.376,A -85,B 0,C 180,E1 22972.039,E2 22972.039} C_VEL
LIN {X 0,Y 474.514,Z 957.008,A -85,B 0,C 180,E1 22969.829,E2 22969.829} C_VEL
LIN {X 0,Y 473.548,Z 968.537,A -85,B 0,C 180,E1 22967.445,E2 22967.445} C_VEL
LIN {X 0,Y 472.832,Z 978.68,A -85,B 0,C 180,E1 22964.949,E2 22964.949} C_VEL
LIN {X 0,Y 472.372,Z 987.056,A -85,B 0,C 180,E1 22962.468,E2 22962.468} C_VEL
LIN {X 0,Y 472.098,Z 993.687,A -85,B 0,C 180,E1 22959.996,E2 22959.996} C_VEL
LIN {X 0,Y 471.956,Z 998.987,A -85,B 0,C 180,E1 22957.425,E2 22957.425} C_VEL
LIN {X 0,Y 471.906,Z 1002.577,A -85,B 0,C 180,E1 22954.983,E2 22954.983} C_VEL
LIN {X 0,Y 471.901,Z 1004.746,A -85,B 0,C 180,E1 22952.429,E2 22952.429} C_VEL
LIN {X 0,Y 471.907,Z 1005.484,A -85,B 0,C 180,E1 22949.879,E2 22949.879} C_VEL
LIN {X 0,Y 471.897,Z 1004.677,A -85,B 0,C 180,E1 22947.45,E2 22947.45} C_VEL
LIN {X 0,Y 471.909,Z 1002.257,A -85,B 0,C 180,E1 22944.774,E2 22944.774} C_VEL
LIN {X 0,Y 471.969,Z 998.573,A -85,B 0,C 180,E1 22942.331,E2 22942.331} C_VEL
LIN {X 0,Y 472.125,Z 993.071,A -85,B 0,C 180,E1 22939.754,E2 22939.754} C_VEL
LIN {X 0,Y 472.415,Z 986.317,A -85,B 0,C 180,E1 22937.286,E2 22937.286} C_VEL
LIN {X 0,Y 472.896,Z 977.763,A -85,B 0,C 180,E1 22934.803,E2 22934.803} C_VEL
LIN {X 0,Y 473.633,Z 967.395,A -85,B 0,C 180,E1 22932.305,E2 22932.305} C_VEL
LIN {X 0,Y 474.635,Z 955.674,A -85,B 0,C 180,E1 22929.92,E2 22929.92} C_VEL
LIN {X 0,Y 475.896,Z 942.483,A -85,B 0,C 180,E1 22927.652,E2 22927.652} C_VEL
LIN {X 0,Y 477.404,Z 927.89,A -85,B 0,C 180,E1 22925.504,E2 22925.504} C_VEL
LIN {X 0,Y 479.165,Z 911.927,A -85,B 0,C 180,E1 22923.481,E2 22923.481} C_VEL
LIN {X 0,Y 480.897,Z 896.196,A -85,B 0,C 180,E1 22921.774,E2 22921.774} C_VEL
LIN {X 0,Y 482.577,Z 878.259,A -85,B 0,C 180,E1 22920.185,E2 22920.185} C_VEL
LIN {X 0,Y 484.317,Z 858.883,A -85,B 0,C 180,E1 22918.725,E2 22918.725} C_VEL
LIN {X 0,Y 485.983,Z 838.737,A -85,B 0,C 180,E1 22917.456,E2 22917.456} C_VEL
LIN {X 0,Y 487.521,Z 817.949,A -85,B 0,C 180,E1 22916.373,E2 22916.373} C_VEL
LIN {X 0,Y 488.968,Z 796.237,A -85,B 0,C 180,E1 22915.464,E2 22915.464} C_VEL
LIN {X 0,Y 490.115,Z 774.514,A -85,B 0,C 180,E1 22914.774,E2 22914.774} C_VEL
LIN {X 0,Y 491.008,Z 752.105,A -85,B 0,C 180,E1 22914.281,E2 22914.281} C_VEL
LIN {X 0,Y 494.724,Z 537.741,A -85,B 0,C 180,E1 22910.813,E2 22910.813} C_VEL
LIN {X 0,Y 495.726,Z 476.183,A -85,B 0,C 180,E1 22909.778,E2 22909.778} C_VEL
LIN {X 0,Y 492.285,Z 450.025,A -85,B 0,C 180,E1 22908.969,E2 22908.969} C_VEL
LIN {X 0,Y 494.168,Z 417.455,A -85,B 0,C 180,E1 22906.858,E2 22906.858} C_VEL
LIN {X 0,Y 484.143,Z 395.251,A -85,B 0,C 180,E1 22904.27,E2 22904.27} C_VEL
LIN {X 0,Y 476.245,Z 379.229,A -85,B 0,C 180,E1 22902.181,E2 22902.181} C_VEL
LIN {X 0,Y 474.648,Z 375.894,A -85,B 0,C 180,E1 22901.733,E2 22901.733} C_VEL
LIN {X 0,Y 472.964,Z 372.292,A -85,B 0,C 180,E1 22901.208,E2 22901.208} C_VEL
LIN {X 0,Y 472.902,Z 371.799,A -85,B 0,C 180,E1 22900.792,E2 22900.792} C_VEL
LIN {X 0,Y 472.886,Z 371.818,A -85,B 0,C 180,E1 22897.208,E2 22897.208} C_VEL
LIN {X 0,Y 472.911,Z 371.824,A -85,B 0,C 180,E1 22893.637,E2 22893.637} C_VEL
LIN {X 0,Y 472.934,Z 371.788,A -85,B 0,C 180,E1 22890.07,E2 22890.07} C_VEL
LIN {X 0,Y 472.881,Z 371.829,A -85,B 0,C 180,E1 22886.631,E2 22886.631} C_VEL
LIN {X 0,Y 472.875,Z 371.806,A -85,B 0,C 180,E1 22882.895,E2 22882.895} C_VEL
LIN {X 0,Y 472.921,Z 371.818,A -85,B 0,C 180,E1 22879.466,E2 22879.466} C_VEL
LIN {X 0,Y 472.893,Z 371.825,A -85,B 0,C 180,E1 22875.954,E2 22875.954} C_VEL
LIN {X 0,Y 472.87,Z 371.828,A -85,B 0,C 180,E1 22872.455,E2 22872.455} C_VEL
LIN {X 0,Y 472.896,Z 371.827,A -85,B 0,C 180,E1 22868.879,E2 22868.879} C_VEL
LIN {X 0,Y 472.92,Z 371.824,A -85,B 0,C 180,E1 22865.459,E2 22865.459} C_VEL
LIN {X 0,Y 472.882,Z 371.821,A -85,B 0,C 180,E1 22861.938,E2 22861.938} C_VEL
LIN {X 0,Y 472.887,Z 371.815,A -85,B 0,C 180,E1 22858.303,E2 22858.303} C_VEL
LIN {X 0,Y 472.937,Z 371.812,A -85,B 0,C 180,E1 22854.784,E2 22854.784} C_VEL
LIN {X 0,Y 472.903,Z 371.827,A -85,B 0,C 180,E1 22851.366,E2 22851.366} C_VEL
LIN {X 0,Y 472.892,Z 371.825,A -85,B 0,C 180,E1 22847.793,E2 22847.793} C_VEL
LIN {X 0,Y 472.929,Z 371.82,A -85,B 0,C 180,E1 22844.299,E2 22844.299} C_VEL
LIN {X 0,Y 472.939,Z 371.814,A -85,B 0,C 180,E1 22840.743,E2 22840.743} C_VEL
LIN {X 0,Y 472.903,Z 371.82,A -85,B 0,C 180,E1 22837.237,E2 22837.237} C_VEL
LIN {X 0,Y 472.905,Z 371.819,A -85,B 0,C 180,E1 22833.505,E2 22833.505} C_VEL
LIN {X 0,Y 472.96,Z 371.813,A -85,B 0,C 180,E1 22830.071,E2 22830.071} C_VEL
LIN {X 0,Y 472.935,Z 371.82,A -85,B 0,C 180,E1 22826.509,E2 22826.509} C_VEL
LIN {X 0,Y 472.91,Z 371.814,A -85,B 0,C 180,E1 22822.946,E2 22822.946} C_VEL
LIN {X 0,Y 472.932,Z 371.815,A -85,B 0,C 180,E1 22819.368,E2 22819.368} C_VEL
LIN {X 0,Y 472.951,Z 371.789,A -85,B 0,C 180,E1 22815.761,E2 22815.761} C_VEL
LIN {X 0,Y 472.931,Z 371.804,A -85,B 0,C 180,E1 22812.24,E2 22812.24} C_VEL
LIN {X 0,Y 472.99,Z 372.08,A -85,B 0,C 180,E1 22809.313,E2 22809.313} C_VEL
LIN {X 0,Y 475.816,Z 378.95,A -85,B 0,C 180,E1 22808.15,E2 22808.15} C_VEL
LIN {X 0,Y 480.422,Z 389.635,A -85,B 0,C 180,E1 22806.524,E2 22806.524} C_VEL
LIN {X 0,Y 493.039,Z 410.266,A -85,B 0,C 180,E1 22804.948,E2 22804.948} C_VEL
LIN {X 0,Y 492.343,Z 453.787,A -85,B 0,C 180,E1 22804.26,E2 22804.26} C_VEL
LIN {X 0,Y 491.412,Z 461.488,A -85,B 0,C 180,E1 22804.212,E2 22804.212} C_VEL
LIN {X 0,Y 486.12,Z 482.041,A -85,B 0,C 180,E1 22804.338,E2 22804.338} C_VEL
LIN {X 0,Y 485.42,Z 488.649,A -85,B 0,C 180,E1 22804.289,E2 22804.289} C_VEL
LIN {X 0,Y 482.841,Z 651.71,A -85,B 0,C 180,E1 22801.717,E2 22801.717} C_VEL
LIN {X 0,Y 482.104,Z 671.825,A -85,B 0,C 180,E1 22801.183,E2 22801.183} C_VEL
LIN {X 0,Y 481.06,Z 690.818,A -85,B 0,C 180,E1 22800.47,E2 22800.47} C_VEL
LIN {X 0,Y 479.738,Z 708.758,A -85,B 0,C 180,E1 22799.597,E2 22799.597} C_VEL
LIN {X 0,Y 478.078,Z 726.946,A -85,B 0,C 180,E1 22798.476,E2 22798.476} C_VEL
LIN {X 0,Y 476.194,Z 744.112,A -85,B 0,C 180,E1 22797.17,E2 22797.17} C_VEL
LIN {X 0,Y 474.217,Z 760.465,A -85,B 0,C 180,E1 22795.673,E2 22795.673} C_VEL
LIN {X 0,Y 472.149,Z 776.455,A -85,B 0,C 180,E1 22793.922,E2 22793.922} C_VEL
LIN {X 0,Y 470.258,Z 790.953,A -85,B 0,C 180,E1 22792.025,E2 22792.025} C_VEL
LIN {X 0,Y 468.53,Z 804.266,A -85,B 0,C 180,E1 22789.962,E2 22789.962} C_VEL
LIN {X 0,Y 467.052,Z 816.461,A -85,B 0,C 180,E1 22787.695,E2 22787.695} C_VEL
LIN {X 0,Y 465.848,Z 827.089,A -85,B 0,C 180,E1 22785.305,E2 22785.305} C_VEL
LIN {X 0,Y 465.041,Z 835.753,A -85,B 0,C 180,E1 22782.919,E2 22782.919} C_VEL
LIN {X 0,Y 464.465,Z 843.043,A -85,B 0,C 180,E1 22780.416,E2 22780.416} C_VEL
LIN {X 0,Y 464.166,Z 848.956,A -85,B 0,C 180,E1 22777.74,E2 22777.74} C_VEL
LIN {X 0,Y 464.003,Z 852.922,A -85,B 0,C 180,E1 22775.192,E2 22775.192} C_VEL
LIN {X 0,Y 463.954,Z 855.297,A -85,B 0,C 180,E1 22772.717,E2 22772.717} C_VEL
LIN {X 0,Y 463.944,Z 856.174,A -85,B 0,C 180,E1 22770.123,E2 22770.123} C_VEL
LIN {X 0,Y 463.945,Z 855.461,A -85,B 0,C 180,E1 22767.529,E2 22767.529} C_VEL
LIN {X 0,Y 464,Z 853.171,A -85,B 0,C 180,E1 22764.931,E2 22764.931} C_VEL
LIN {X 0,Y 464.154,Z 849.146,A -85,B 0,C 180,E1 22762.27,E2 22762.27} C_VEL
LIN {X 0,Y 464.441,Z 843.545,A -85,B 0,C 180,E1 22759.686,E2 22759.686} C_VEL
LIN {X 0,Y 464.982,Z 836.472,A -85,B 0,C 180,E1 22757.205,E2 22757.205} C_VEL
LIN {X 0,Y 465.817,Z 827.461,A -85,B 0,C 180,E1 22754.693,E2 22754.693} C_VEL
LIN {X 0,Y 466.997,Z 816.896,A -85,B 0,C 180,E1 22752.302,E2 22752.302} C_VEL
LIN {X 0,Y 468.462,Z 804.76,A -85,B 0,C 180,E1 22750.034,E2 22750.034} C_VEL
LIN {X 0,Y 470.132,Z 791.831,A -85,B 0,C 180,E1 22748.014,E2 22748.014} C_VEL
LIN {X 0,Y 471.987,Z 777.661,A -85,B 0,C 180,E1 22746.135,E2 22746.135} C_VEL
LIN {X 0,Y 474.046,Z 761.913,A -85,B 0,C 180,E1 22744.383,E2 22744.383} C_VEL
LIN {X 0,Y 476.003,Z 745.88,A -85,B 0,C 180,E1 22742.885,E2 22742.885} C_VEL
LIN {X 0,Y 477.869,Z 729.012,A -85,B 0,C 180,E1 22741.578,E2 22741.578} C_VEL
LIN {X 0,Y 479.508,Z 711.257,A -85,B 0,C 180,E1 22740.455,E2 22740.455} C_VEL
LIN {X 0,Y 480.987,Z 691.955,A -85,B 0,C 180,E1 22739.49,E2 22739.49} C_VEL
LIN {X 0,Y 482.072,Z 672.721,A -85,B 0,C 180,E1 22738.755,E2 22738.755} C_VEL
LIN {X 0,Y 482.835,Z 652.35,A -85,B 0,C 180,E1 22738.205,E2 22738.205} C_VEL
LIN {X 0,Y 484.255,Z 562.493,A -85,B 0,C 180,E1 22736.774,E2 22736.774} C_VEL
LIN {X 0,Y 486.599,Z 413.106,A -85,B 0,C 180,E1 22734.408,E2 22734.408} C_VEL
LIN {X 0,Y 474.04,Z 392.87,A -85,B 0,C 180,E1 22732.797,E2 22732.797} C_VEL
LIN {X 0,Y 472.03,Z 389.59,A -85,B 0,C 180,E1 22732.493,E2 22732.493} C_VEL
LIN {X 0,Y 466.178,Z 376.069,A -85,B 0,C 180,E1 22730.276,E2 22730.276} C_VEL
LIN {X 0,Y 465.029,Z 373.031,A -85,B 0,C 180,E1 22729.719,E2 22729.719} C_VEL
LIN {X 0,Y 465.014,Z 372.813,A -85,B 0,C 180,E1 22726.359,E2 22726.359} C_VEL
LIN {X 0,Y 464.994,Z 372.799,A -85,B 0,C 180,E1 22722.666,E2 22722.666} C_VEL
LIN {X 0,Y 464.975,Z 372.775,A -85,B 0,C 180,E1 22719.054,E2 22719.054} C_VEL
LIN {X 0,Y 464.997,Z 372.814,A -85,B 0,C 180,E1 22715.426,E2 22715.426} C_VEL
LIN {X 0,Y 465.018,Z 372.81,A -85,B 0,C 180,E1 22711.789,E2 22711.789} C_VEL
LIN {X 0,Y 464.992,Z 372.812,A -85,B 0,C 180,E1 22708.173,E2 22708.173} C_VEL
LIN {X 0,Y 464.968,Z 372.812,A -85,B 0,C 180,E1 22704.56,E2 22704.56} C_VEL
LIN {X 0,Y 464.977,Z 372.813,A -85,B 0,C 180,E1 22700.914,E2 22700.914} C_VEL
LIN {X 0,Y 465.013,Z 372.81,A -85,B 0,C 180,E1 22697.333,E2 22697.333} C_VEL
LIN {X 0,Y 464.977,Z 372.807,A -85,B 0,C 180,E1 22693.809,E2 22693.809} C_VEL
LIN {X 0,Y 464.955,Z 372.805,A -85,B 0,C 180,E1 22690.282,E2 22690.282} C_VEL
LIN {X 0,Y 464.987,Z 372.802,A -85,B 0,C 180,E1 22686.792,E2 22686.792} C_VEL
LIN {X 0,Y 464.993,Z 372.815,A -85,B 0,C 180,E1 22683.205,E2 22683.205} C_VEL
LIN {X 0,Y 464.948,Z 372.816,A -85,B 0,C 180,E1 22679.754,E2 22679.754} C_VEL
LIN {X 0,Y 464.949,Z 372.816,A -85,B 0,C 180,E1 22676.054,E2 22676.054} C_VEL
LIN {X 0,Y 464.997,Z 372.803,A -85,B 0,C 180,E1 22672.588,E2 22672.588} C_VEL
LIN {X 0,Y 464.962,Z 372.807,A -85,B 0,C 180,E1 22668.967,E2 22668.967} C_VEL
LIN {X 0,Y 464.932,Z 372.814,A -85,B 0,C 180,E1 22665.427,E2 22665.427} C_VEL
LIN {X 0,Y 464.944,Z 372.812,A -85,B 0,C 180,E1 22661.831,E2 22661.831} C_VEL
LIN {X 0,Y 464.997,Z 372.806,A -85,B 0,C 180,E1 22658.252,E2 22658.252} C_VEL
LIN {X 0,Y 464.954,Z 372.787,A -85,B 0,C 180,E1 22654.664,E2 22654.664} C_VEL
LIN {X 0,Y 464.94,Z 372.805,A -85,B 0,C 180,E1 22651.203,E2 22651.203} C_VEL
LIN {X 0,Y 464.977,Z 372.807,A -85,B 0,C 180,E1 22647.673,E2 22647.673} C_VEL
LIN {X 0,Y 464.989,Z 372.779,A -85,B 0,C 180,E1 22644.054,E2 22644.054} C_VEL
LIN {X 0,Y 464.948,Z 372.791,A -85,B 0,C 180,E1 22640.626,E2 22640.626} C_VEL
LIN {X 0,Y 465.053,Z 373.072,A -85,B 0,C 180,E1 22639.718,E2 22639.718} C_VEL
LIN {X 0,Y 466.509,Z 376.614,A -85,B 0,C 180,E1 22639.179,E2 22639.179} C_VEL
LIN {X 0,Y 472.003,Z 387.436,A -85,B 0,C 180,E1 22637.653,E2 22637.653} C_VEL
LIN {X 0,Y 480.238,Z 404.484,A -85,B 0,C 180,E1 22635.442,E2 22635.442} C_VEL
LIN {X 0,Y 487.461,Z 421.184,A -85,B 0,C 180,E1 22633.5,E2 22633.5} C_VEL
LIN {X 0,Y 485.741,Z 450.546,A -85,B 0,C 180,E1 22631.596,E2 22631.596} C_VEL
LIN {X 0,Y 489.43,Z 480.108,A -85,B 0,C 180,E1 22630.699,E2 22630.699} C_VEL
LIN {X 0,Y 485.115,Z 699.432,A -85,B 0,C 180,E1 22627.067,E2 22627.067} C_VEL
LIN {X 0,Y 483.878,Z 758.714,A -85,B 0,C 180,E1 22626.071,E2 22626.071} C_VEL
LIN {X 0,Y 482.778,Z 781.043,A -85,B 0,C 180,E1 22625.494,E2 22625.494} C_VEL
LIN {X 0,Y 481.424,Z 802.667,A -85,B 0,C 180,E1 22624.724,E2 22624.724} C_VEL
LIN {X 0,Y 479.877,Z 823.812,A -85,B 0,C 180,E1 22623.763,E2 22623.763} C_VEL
LIN {X 0,Y 478.104,Z 844.967,A -85,B 0,C 180,E1 22622.564,E2 22622.564} C_VEL
LIN {X 0,Y 476.325,Z 864.48,A -85,B 0,C 180,E1 22621.227,E2 22621.227} C_VEL
LIN {X 0,Y 474.49,Z 883.732,A -85,B 0,C 180,E1 22619.68,E2 22619.68} C_VEL
LIN {X 0,Y 472.579,Z 902.865,A -85,B 0,C 180,E1 22617.875,E2 22617.875} C_VEL
LIN {X 0,Y 471.029,Z 918.017,A -85,B 0,C 180,E1 22616.199,E2 22616.199} C_VEL
LIN {X 0,Y 469.674,Z 929.923,A -85,B 0,C 180,E1 22614.632,E2 22614.632} C_VEL
LIN {X 0,Y 468.009,Z 944.788,A -85,B 0,C 180,E1 22612.349,E2 22612.349} C_VEL
LIN {X 0,Y 466.701,Z 957.646,A -85,B 0,C 180,E1 22610.045,E2 22610.045} C_VEL
LIN {X 0,Y 465.65,Z 969.353,A -85,B 0,C 180,E1 22607.567,E2 22607.567} C_VEL
LIN {X 0,Y 464.892,Z 979.235,A -85,B 0,C 180,E1 22605.056,E2 22605.056} C_VEL
LIN {X 0,Y 464.382,Z 987.764,A -85,B 0,C 180,E1 22602.433,E2 22602.433} C_VEL
LIN {X 0,Y 464.1,Z 994.281,A -85,B 0,C 180,E1 22599.924,E2 22599.924} C_VEL
LIN {X 0,Y 463.959,Z 999.193,A -85,B 0,C 180,E1 22597.429,E2 22597.429} C_VEL
LIN {X 0,Y 463.907,Z 1002.736,A -85,B 0,C 180,E1 22594.946,E2 22594.946} C_VEL
LIN {X 0,Y 463.904,Z 1004.814,A -85,B 0,C 180,E1 22592.347,E2 22592.347} C_VEL
LIN {X 0,Y 463.9,Z 1005.462,A -85,B 0,C 180,E1 22589.753,E2 22589.753} C_VEL
LIN {X 0,Y 463.895,Z 1004.609,A -85,B 0,C 180,E1 22587.283,E2 22587.283} C_VEL
LIN {X 0,Y 463.918,Z 1002.097,A -85,B 0,C 180,E1 22584.559,E2 22584.559} C_VEL
LIN {X 0,Y 463.995,Z 998.366,A -85,B 0,C 180,E1 22582.074,E2 22582.074} C_VEL
LIN {X 0,Y 464.171,Z 992.768,A -85,B 0,C 180,E1 22579.451,E2 22579.451} C_VEL
LIN {X 0,Y 464.513,Z 985.506,A -85,B 0,C 180,E1 22576.813,E2 22576.813} C_VEL
LIN {X 0,Y 465.067,Z 976.843,A -85,B 0,C 180,E1 22574.285,E2 22574.285} C_VEL
LIN {X 0,Y 465.854,Z 966.82,A -85,B 0,C 180,E1 22571.87,E2 22571.87} C_VEL
LIN {X 0,Y 466.965,Z 954.972,A -85,B 0,C 180,E1 22569.445,E2 22569.445} C_VEL
LIN {X 0,Y 468.365,Z 941.711,A -85,B 0,C 180,E1 22567.14,E2 22567.14} C_VEL
LIN {X 0,Y 470.022,Z 926.963,A -85,B 0,C 180,E1 22564.959,E2 22564.959} C_VEL
LIN {X 0,Y 471.421,Z 914.439,A -85,B 0,C 180,E1 22563.373,E2 22563.373} C_VEL
LIN {X 0,Y 473.191,Z 896.749,A -85,B 0,C 180,E1 22561.523,E2 22561.523} C_VEL
LIN {X 0,Y 475.154,Z 876.638,A -85,B 0,C 180,E1 22559.721,E2 22559.721} C_VEL
LIN {X 0,Y 476.993,Z 857.447,A -85,B 0,C 180,E1 22558.259,E2 22558.259} C_VEL
LIN {X 0,Y 478.767,Z 837.296,A -85,B 0,C 180,E1 22556.975,E2 22556.975} C_VEL
LIN {X 0,Y 480.482,Z 815.954,A -85,B 0,C 180,E1 22555.856,E2 22555.856} C_VEL
LIN {X 0,Y 481.986,Z 794.117,A -85,B 0,C 180,E1 22554.943,E2 22554.943} C_VEL
LIN {X 0,Y 483.273,Z 771.824,A -85,B 0,C 180,E1 22554.239,E2 22554.239} C_VEL
LIN {X 0,Y 484.168,Z 749.63,A -85,B 0,C 180,E1 22553.76,E2 22553.76} C_VEL
LIN {X 0,Y 488.322,Z 532.592,A -85,B 0,C 180,E1 22550.18,E2 22550.18} C_VEL
LIN {X 0,Y 489.306,Z 477.576,A -85,B 0,C 180,E1 22549.241,E2 22549.241} C_VEL
LIN {X 0,Y 485.674,Z 449.43,A -85,B 0,C 180,E1 22548.357,E2 22548.357} C_VEL
LIN {X 0,Y 487.436,Z 420.909,A -85,B 0,C 180,E1 22546.478,E2 22546.478} C_VEL
LIN {X 0,Y 478.03,Z 399.862,A -85,B 0,C 180,E1 22543.981,E2 22543.981} C_VEL
LIN {X 0,Y 469.055,Z 381.378,A -85,B 0,C 180,E1 22541.524,E2 22541.524} C_VEL
LIN {X 0,Y 465.142,Z 373.591,A -85,B 0,C 180,E1 22540.398,E2 22540.398} C_VEL
LIN {X 0,Y 465.015,Z 372.823,A -85,B 0,C 180,E1 22540.169,E2 22540.169} C_VEL
LIN {X 0,Y 464.968,Z 372.788,A -85,B 0,C 180,E1 22536.559,E2 22536.559} C_VEL
LIN {X 0,Y 464.946,Z 372.82,A -85,B 0,C 180,E1 22532.961,E2 22532.961} C_VEL
LIN {X 0,Y 464.954,Z 372.788,A -85,B 0,C 180,E1 22529.36,E2 22529.36} C_VEL
LIN {X 0,Y 464.992,Z 372.792,A -85,B 0,C 180,E1 22525.881,E2 22525.881} C_VEL
LIN {X 0,Y 464.943,Z 372.805,A -85,B 0,C 180,E1 22522.373,E2 22522.373} C_VEL
LIN {X 0,Y 464.935,Z 372.81,A -85,B 0,C 180,E1 22518.819,E2 22518.819} C_VEL
LIN {X 0,Y 464.978,Z 372.805,A -85,B 0,C 180,E1 22515.336,E2 22515.336} C_VEL
LIN {X 0,Y 464.96,Z 372.81,A -85,B 0,C 180,E1 22511.788,E2 22511.788} C_VEL
LIN {X 0,Y 464.934,Z 372.816,A -85,B 0,C 180,E1 22508.284,E2 22508.284} C_VEL
LIN {X 0,Y 464.956,Z 372.816,A -85,B 0,C 180,E1 22504.687,E2 22504.687} C_VEL
LIN {X 0,Y 465.004,Z 372.812,A -85,B 0,C 180,E1 22501.109,E2 22501.109} C_VEL
LIN {X 0,Y 464.96,Z 372.805,A -85,B 0,C 180,E1 22497.535,E2 22497.535} C_VEL
LIN {X 0,Y 464.946,Z 372.802,A -85,B 0,C 180,E1 22493.951,E2 22493.951} C_VEL
LIN {X 0,Y 464.983,Z 372.804,A -85,B 0,C 180,E1 22490.469,E2 22490.469} C_VEL
LIN {X 0,Y 465.006,Z 372.811,A -85,B 0,C 180,E1 22486.825,E2 22486.825} C_VEL
LIN {X 0,Y 464.96,Z 372.815,A -85,B 0,C 180,E1 22483.381,E2 22483.381} C_VEL
LIN {X 0,Y 464.962,Z 372.813,A -85,B 0,C 180,E1 22479.632,E2 22479.632} C_VEL
LIN {X 0,Y 465.001,Z 372.806,A -85,B 0,C 180,E1 22476.156,E2 22476.156} C_VEL
LIN {X 0,Y 465.009,Z 372.803,A -85,B 0,C 180,E1 22472.465,E2 22472.465} C_VEL
LIN {X 0,Y 464.971,Z 372.805,A -85,B 0,C 180,E1 22468.929,E2 22468.929} C_VEL
LIN {X 0,Y 464.971,Z 372.811,A -85,B 0,C 180,E1 22465.22,E2 22465.22} C_VEL
LIN {X 0,Y 465.005,Z 372.772,A -85,B 0,C 180,E1 22461.697,E2 22461.697} C_VEL
LIN {X 0,Y 465.014,Z 372.81,A -85,B 0,C 180,E1 22458.033,E2 22458.033} C_VEL
LIN {X 0,Y 464.983,Z 372.794,A -85,B 0,C 180,E1 22454.446,E2 22454.446} C_VEL
LIN {X 0,Y 464.979,Z 372.783,A -85,B 0,C 180,E1 22450.806,E2 22450.806} C_VEL
LIN {X 0,Y 465.045,Z 373.127,A -85,B 0,C 180,E1 22450.152,E2 22450.152} C_VEL
LIN {X 0,Y 471.663,Z 388.704,A -85,B 0,C 180,E1 22447.549,E2 22447.549} C_VEL
LIN {X 0,Y 472.946,Z 391.163,A -85,B 0,C 180,E1 22447.254,E2 22447.254} C_VEL
LIN {X 0,Y 486.102,Z 412.269,A -85,B 0,C 180,E1 22445.56,E2 22445.56} C_VEL
LIN {X 0,Y 486.728,Z 413.817,A -85,B 0,C 180,E1 22445.473,E2 22445.473} C_VEL
LIN {X 0,Y 485.42,Z 488.649,A -85,B 0,C 180,E1 22444.289,E2 22444.289} C_VEL
LIN {X 0,Y 484.498,Z 496.351,A -85,B 0,C 180,E1 22444.24,E2 22444.24} C_VEL
LIN {X 0,Y 479.17,Z 516.895,A -85,B 0,C 180,E1 22444.375,E2 22444.375} C_VEL
LIN {X 0,Y 478.48,Z 523.503,A -85,B 0,C 180,E1 22444.324,E2 22444.324} C_VEL
LIN {X 0,Y 476.338,Z 653.019,A -85,B 0,C 180,E1 22442.257,E2 22442.257} C_VEL
LIN {X 0,Y 475.573,Z 673.191,A -85,B 0,C 180,E1 22441.714,E2 22441.714} C_VEL
LIN {X 0,Y 474.459,Z 692.562,A -85,B 0,C 180,E1 22440.975,E2 22440.975} C_VEL
LIN {X 0,Y 473.025,Z 711,A -85,B 0,C 180,E1 22440.06,E2 22440.06} C_VEL
LIN {X 0,Y 471.314,Z 729.186,A -85,B 0,C 180,E1 22438.923,E2 22438.923} C_VEL
LIN {X 0,Y 469.353,Z 746.307,A -85,B 0,C 180,E1 22437.6,E2 22437.6} C_VEL
LIN {X 0,Y 467.271,Z 762.565,A -85,B 0,C 180,E1 22436.083,E2 22436.083} C_VEL
LIN {X 0,Y 464.994,Z 778.934,A -85,B 0,C 180,E1 22434.246,E2 22434.246} C_VEL
LIN {X 0,Y 462.991,Z 793.139,A -85,B 0,C 180,E1 22432.336,E2 22432.336} C_VEL
LIN {X 0,Y 461.169,Z 805.974,A -85,B 0,C 180,E1 22430.295,E2 22430.295} C_VEL
LIN {X 0,Y 459.556,Z 818.067,A -85,B 0,C 180,E1 22427.994,E2 22427.994} C_VEL
LIN {X 0,Y 458.237,Z 828.623,A -85,B 0,C 180,E1 22425.566,E2 22425.566} C_VEL
LIN {X 0,Y 457.338,Z 837.226,A -85,B 0,C 180,E1 22423.141,E2 22423.141} C_VEL
LIN {X 0,Y 456.681,Z 844.545,A -85,B 0,C 180,E1 22420.566,E2 22420.566} C_VEL
LIN {X 0,Y 456.341,Z 850.235,A -85,B 0,C 180,E1 22417.933,E2 22417.933} C_VEL
LIN {X 0,Y 456.136,Z 854.276,A -85,B 0,C 180,E1 22415.281,E2 22415.281} C_VEL
LIN {X 0,Y 456.07,Z 856.631,A -85,B 0,C 180,E1 22412.764,E2 22412.764} C_VEL
LIN {X 0,Y 456.055,Z 857.502,A -85,B 0,C 180,E1 22410.125,E2 22410.125} C_VEL
LIN {X 0,Y 456.06,Z 856.795,A -85,B 0,C 180,E1 22407.487,E2 22407.487} C_VEL
LIN {X 0,Y 456.132,Z 854.526,A -85,B 0,C 180,E1 22404.844,E2 22404.844} C_VEL
LIN {X 0,Y 456.317,Z 850.63,A -85,B 0,C 180,E1 22402.193,E2 22402.193} C_VEL
LIN {X 0,Y 456.635,Z 845.336,A -85,B 0,C 180,E1 22399.657,E2 22399.657} C_VEL
LIN {X 0,Y 457.237,Z 838.358,A -85,B 0,C 180,E1 22397.113,E2 22397.113} C_VEL
LIN {X 0,Y 458.145,Z 829.482,A -85,B 0,C 180,E1 22394.56,E2 22394.56} C_VEL
LIN {X 0,Y 459.411,Z 819.057,A -85,B 0,C 180,E1 22392.131,E2 22392.131} C_VEL
LIN {X 0,Y 460.892,Z 807.795,A -85,B 0,C 180,E1 22389.943,E2 22389.943} C_VEL
LIN {X 0,Y 462.777,Z 794.557,A -85,B 0,C 180,E1 22387.786,E2 22387.786} C_VEL
LIN {X 0,Y 464.901,Z 779.615,A -85,B 0,C 180,E1 22385.748,E2 22385.748} C_VEL
LIN {X 0,Y 467.096,Z 764.008,A -85,B 0,C 180,E1 22383.974,E2 22383.974} C_VEL
LIN {X 0,Y 469.179,Z 747.892,A -85,B 0,C 180,E1 22382.441,E2 22382.441} C_VEL
LIN {X 0,Y 471.187,Z 730.305,A -85,B 0,C 180,E1 22381.068,E2 22381.068} C_VEL
LIN {X 0,Y 472.895,Z 712.404,A -85,B 0,C 180,E1 22379.93,E2 22379.93} C_VEL
LIN {X 0,Y 474.436,Z 692.957,A -85,B 0,C 180,E1 22378.952,E2 22378.952} C_VEL
LIN {X 0,Y 475.559,Z 673.611,A -85,B 0,C 180,E1 22378.209,E2 22378.209} C_VEL
LIN {X 0,Y 476.339,Z 653.272,A -85,B 0,C 180,E1 22377.657,E2 22377.657} C_VEL
LIN {X 0,Y 478.062,Z 549.408,A -85,B 0,C 180,E1 22375.993,E2 22375.993} C_VEL
LIN {X 0,Y 480.362,Z 416.278,A -85,B 0,C 180,E1 22373.863,E2 22373.863} C_VEL
LIN {X 0,Y 467.323,Z 395.375,A -85,B 0,C 180,E1 22372.138,E2 22372.138} C_VEL
LIN {X 0,Y 464.101,Z 390.277,A -85,B 0,C 180,E1 22371.647,E2 22371.647} C_VEL
LIN {X 0,Y 458.488,Z 377.46,A -85,B 0,C 180,E1 22369.473,E2 22369.473} C_VEL
LIN {X 0,Y 457.09,Z 373.984,A -85,B 0,C 180,E1 22368.806,E2 22368.806} C_VEL
LIN {X 0,Y 457.042,Z 373.775,A -85,B 0,C 180,E1 22365.138,E2 22365.138} C_VEL
LIN {X 0,Y 457.049,Z 373.805,A -85,B 0,C 180,E1 22361.384,E2 22361.384} C_VEL
LIN {X 0,Y 457.071,Z 373.764,A -85,B 0,C 180,E1 22357.772,E2 22357.772} C_VEL
LIN {X 0,Y 457.07,Z 373.792,A -85,B 0,C 180,E1 22354.057,E2 22354.057} C_VEL
LIN {X 0,Y 457.04,Z 373.791,A -85,B 0,C 180,E1 22350.473,E2 22350.473} C_VEL
LIN {X 0,Y 457.031,Z 373.794,A -85,B 0,C 180,E1 22346.787,E2 22346.787} C_VEL
LIN {X 0,Y 457.055,Z 373.79,A -85,B 0,C 180,E1 22343.19,E2 22343.19} C_VEL
LIN {X 0,Y 457.072,Z 373.789,A -85,B 0,C 180,E1 22339.554,E2 22339.554} C_VEL
LIN {X 0,Y 457.033,Z 373.801,A -85,B 0,C 180,E1 22336.001,E2 22336.001} C_VEL
LIN {X 0,Y 457.02,Z 373.804,A -85,B 0,C 180,E1 22332.381,E2 22332.381} C_VEL
LIN {X 0,Y 457.046,Z 373.804,A -85,B 0,C 180,E1 22328.809,E2 22328.809} C_VEL
LIN {X 0,Y 457.056,Z 373.789,A -85,B 0,C 180,E1 22325.272,E2 22325.272} C_VEL
LIN {X 0,Y 457.017,Z 373.791,A -85,B 0,C 180,E1 22321.63,E2 22321.63} C_VEL
LIN {X 0,Y 457.006,Z 373.798,A -85,B 0,C 180,E1 22317.994,E2 22317.994} C_VEL
LIN {X 0,Y 457.037,Z 373.802,A -85,B 0,C 180,E1 22314.448,E2 22314.448} C_VEL
LIN {X 0,Y 457.036,Z 373.804,A -85,B 0,C 180,E1 22310.938,E2 22310.938} C_VEL
LIN {X 0,Y 457,Z 373.805,A -85,B 0,C 180,E1 22307.343,E2 22307.343} C_VEL
LIN {X 0,Y 456.994,Z 373.808,A -85,B 0,C 180,E1 22303.606,E2 22303.606} C_VEL
LIN {X 0,Y 457.029,Z 373.803,A -85,B 0,C 180,E1 22300.045,E2 22300.045} C_VEL
LIN {X 0,Y 457.028,Z 373.765,A -85,B 0,C 180,E1 22296.537,E2 22296.537} C_VEL
LIN {X 0,Y 457.003,Z 373.809,A -85,B 0,C 180,E1 22292.931,E2 22292.931} C_VEL
LIN {X 0,Y 457.001,Z 373.77,A -85,B 0,C 180,E1 22289.206,E2 22289.206} C_VEL
LIN {X 0,Y 457.041,Z 373.782,A -85,B 0,C 180,E1 22285.638,E2 22285.638} C_VEL
LIN {X 0,Y 457.067,Z 373.803,A -85,B 0,C 180,E1 22281.911,E2 22281.911} C_VEL
LIN {X 0,Y 457.028,Z 373.926,A -85,B 0,C 180,E1 22280.711,E2 22280.711} C_VEL
LIN {X 0,Y 457.414,Z 375.457,A -85,B 0,C 180,E1 22280.418,E2 22280.418} C_VEL
LIN {X 0,Y 459.704,Z 379.692,A -85,B 0,C 180,E1 22279.761,E2 22279.761} C_VEL
LIN {X 0,Y 467.691,Z 395.438,A -85,B 0,C 180,E1 22277.502,E2 22277.502} C_VEL
LIN {X 0,Y 476.966,Z 415.567,A -85,B 0,C 180,E1 22274.942,E2 22274.942} C_VEL
LIN {X 0,Y 480.79,Z 424.483,A -85,B 0,C 180,E1 22273.897,E2 22273.897} C_VEL
LIN {X 0,Y 479.186,Z 449.852,A -85,B 0,C 180,E1 22272.23,E2 22272.23} C_VEL
LIN {X 0,Y 483.049,Z 481.302,A -85,B 0,C 180,E1 22271.255,E2 22271.255} C_VEL
LIN {X 0,Y 478.266,Z 703.12,A -85,B 0,C 180,E1 22267.514,E2 22267.514} C_VEL
LIN {X 0,Y 477.014,Z 757.676,A -85,B 0,C 180,E1 22266.577,E2 22266.577} C_VEL
LIN {X 0,Y 475.813,Z 780.169,A -85,B 0,C 180,E1 22265.985,E2 22265.985} C_VEL
LIN {X 0,Y 474.318,Z 802.316,A -85,B 0,C 180,E1 22265.181,E2 22265.181} C_VEL
LIN {X 0,Y 472.6,Z 823.993,A -85,B 0,C 180,E1 22264.171,E2 22264.171} C_VEL
LIN {X 0,Y 470.723,Z 845.376,A -85,B 0,C 180,E1 22262.937,E2 22262.937} C_VEL
LIN {X 0,Y 468.849,Z 864.537,A -85,B 0,C 180,E1 22261.589,E2 22261.589} C_VEL
LIN {X 0,Y 466.807,Z 884.486,A -85,B 0,C 180,E1 22259.935,E2 22259.935} C_VEL
LIN {X 0,Y 464.939,Z 902.126,A -85,B 0,C 180,E1 22258.234,E2 22258.234} C_VEL
LIN {X 0,Y 463.084,Z 919.464,A -85,B 0,C 180,E1 22256.269,E2 22256.269} C_VEL
LIN {X 0,Y 461.397,Z 935.453,A -85,B 0,C 180,E1 22254.173,E2 22254.173} C_VEL
LIN {X 0,Y 460.388,Z 944.783,A -85,B 0,C 180,E1 22252.74,E2 22252.74} C_VEL
LIN {X 0,Y 458.966,Z 957.645,A -85,B 0,C 180,E1 22250.398,E2 22250.398} C_VEL
LIN {X 0,Y 457.84,Z 969.107,A -85,B 0,C 180,E1 22247.933,E2 22247.933} C_VEL
LIN {X 0,Y 457.002,Z 979.137,A -85,B 0,C 180,E1 22245.35,E2 22245.35} C_VEL
LIN {X 0,Y 456.436,Z 987.764,A -85,B 0,C 180,E1 22242.653,E2 22242.653} C_VEL
LIN {X 0,Y 456.125,Z 994.281,A -85,B 0,C 180,E1 22240.099,E2 22240.099} C_VEL
LIN {X 0,Y 455.967,Z 999.193,A -85,B 0,C 180,E1 22237.56,E2 22237.56} C_VEL
LIN {X 0,Y 455.908,Z 1002.736,A -85,B 0,C 180,E1 22235.033,E2 22235.033} C_VEL
LIN {X 0,Y 455.903,Z 1004.814,A -85,B 0,C 180,E1 22232.388,E2 22232.388} C_VEL
LIN {X 0,Y 455.9,Z 1005.462,A -85,B 0,C 180,E1 22229.749,E2 22229.749} C_VEL
LIN {X 0,Y 455.895,Z 1004.608,A -85,B 0,C 180,E1 22227.235,E2 22227.235} C_VEL
LIN {X 0,Y 455.925,Z 1002.097,A -85,B 0,C 180,E1 22224.464,E2 22224.464} C_VEL
LIN {X 0,Y 456.01,Z 998.366,A -85,B 0,C 180,E1 22221.934,E2 22221.934} C_VEL
LIN {X 0,Y 456.199,Z 992.768,A -85,B 0,C 180,E1 22219.265,E2 22219.265} C_VEL
LIN {X 0,Y 456.575,Z 985.506,A -85,B 0,C 180,E1 22216.579,E2 22216.579} C_VEL
LIN {X 0,Y 457.185,Z 976.843,A -85,B 0,C 180,E1 22214.007,E2 22214.007} C_VEL
LIN {X 0,Y 458.044,Z 966.819,A -85,B 0,C 180,E1 22211.55,E2 22211.55} C_VEL
LIN {X 0,Y 459.262,Z 954.856,A -85,B 0,C 180,E1 22209.062,E2 22209.062} C_VEL
LIN {X 0,Y 460.663,Z 942.433,A -85,B 0,C 180,E1 22206.871,E2 22206.871} C_VEL
LIN {X 0,Y 462.155,Z 928.142,A -85,B 0,C 180,E1 22204.83,E2 22204.83} C_VEL
LIN {X 0,Y 463.904,Z 911.737,A -85,B 0,C 180,E1 22202.815,E2 22202.815} C_VEL
LIN {X 0,Y 465.858,Z 893.604,A -85,B 0,C 180,E1 22200.914,E2 22200.914} C_VEL
LIN {X 0,Y 467.806,Z 874.81,A -85,B 0,C 180,E1 22199.227,E2 22199.227} C_VEL
LIN {X 0,Y 469.784,Z 855.055,A -85,B 0,C 180,E1 22197.714,E2 22197.714} C_VEL
LIN {X 0,Y 471.697,Z 834.641,A -85,B 0,C 180,E1 22196.412,E2 22196.412} C_VEL
LIN {X 0,Y 473.463,Z 813.546,A -85,B 0,C 180,E1 22195.315,E2 22195.315} C_VEL
LIN {X 0,Y 475.109,Z 790.623,A -85,B 0,C 180,E1 22194.366,E2 22194.366} C_VEL
LIN {X 0,Y 476.495,Z 768.595,A -85,B 0,C 180,E1 22193.682,E2 22193.682} C_VEL
LIN {X 0,Y 477.41,Z 745.955,A -85,B 0,C 180,E1 22193.201,E2 22193.201} C_VEL
LIN {X 0,Y 481.949,Z 529.528,A -85,B 0,C 180,E1 22189.564,E2 22189.564} C_VEL
LIN {X 0,Y 482.916,Z 478.822,A -85,B 0,C 180,E1 22188.684,E2 22188.684} C_VEL
LIN {X 0,Y 479.131,Z 448.468,A -85,B 0,C 180,E1 22187.707,E2 22187.707} C_VEL
LIN {X 0,Y 480.785,Z 424.477,A -85,B 0,C 180,E1 22186.103,E2 22186.103} C_VEL
LIN {X 0,Y 472.37,Z 405.352,A -85,B 0,C 180,E1 22183.801,E2 22183.801} C_VEL
LIN {X 0,Y 463.468,Z 386.85,A -85,B 0,C 180,E1 22181.311,E2 22181.311} C_VEL
LIN {X 0,Y 458.899,Z 377.963,A -85,B 0,C 180,E1 22179.997,E2 22179.997} C_VEL
LIN {X 0,Y 457.151,Z 374.551,A -85,B 0,C 180,E1 22179.468,E2 22179.468} C_VEL
LIN {X 0,Y 457.012,Z 373.813,A -85,B 0,C 180,E1 22179.218,E2 22179.218} C_VEL
LIN {X 0,Y 457.022,Z 373.769,A -85,B 0,C 180,E1 22175.587,E2 22175.587} C_VEL
LIN {X 0,Y 457.062,Z 373.782,A -85,B 0,C 180,E1 22171.964,E2 22171.964} C_VEL
LIN {X 0,Y 457.017,Z 373.798,A -85,B 0,C 180,E1 22168.43,E2 22168.43} C_VEL
LIN {X 0,Y 456.994,Z 373.766,A -85,B 0,C 180,E1 22164.786,E2 22164.786} C_VEL
LIN {X 0,Y 457.014,Z 373.809,A -85,B 0,C 180,E1 22161.161,E2 22161.161} C_VEL
LIN {X 0,Y 457.049,Z 373.804,A -85,B 0,C 180,E1 22157.502,E2 22157.502} C_VEL
LIN {X 0,Y 457.013,Z 373.803,A -85,B 0,C 180,E1 22153.925,E2 22153.925} C_VEL
LIN {X 0,Y 456.996,Z 373.802,A -85,B 0,C 180,E1 22150.335,E2 22150.335} C_VEL
LIN {X 0,Y 457.009,Z 373.797,A -85,B 0,C 180,E1 22146.658,E2 22146.658} C_VEL
LIN {X 0,Y 457.054,Z 373.79,A -85,B 0,C 180,E1 22143.135,E2 22143.135} C_VEL
LIN {X 0,Y 457.018,Z 373.805,A -85,B 0,C 180,E1 22139.624,E2 22139.624} C_VEL
LIN {X 0,Y 457.007,Z 373.805,A -85,B 0,C 180,E1 22135.985,E2 22135.985} C_VEL
LIN {X 0,Y 457.027,Z 373.803,A -85,B 0,C 180,E1 22132.331,E2 22132.331} C_VEL
LIN {X 0,Y 457.066,Z 373.79,A -85,B 0,C 180,E1 22128.773,E2 22128.773} C_VEL
LIN {X 0,Y 457.032,Z 373.792,A -85,B 0,C 180,E1 22125.169,E2 22125.169} C_VEL
LIN {X 0,Y 457.021,Z 373.799,A -85,B 0,C 180,E1 22121.504,E2 22121.504} C_VEL
LIN {X 0,Y 457.037,Z 373.798,A -85,B 0,C 180,E1 22117.896,E2 22117.896} C_VEL
LIN {X 0,Y 457.073,Z 373.797,A -85,B 0,C 180,E1 22114.311,E2 22114.311} C_VEL
LIN {X 0,Y 457.053,Z 373.803,A -85,B 0,C 180,E1 22110.657,E2 22110.657} C_VEL
LIN {X 0,Y 457.03,Z 373.805,A -85,B 0,C 180,E1 22107.14,E2 22107.14} C_VEL
LIN {X 0,Y 457.048,Z 373.799,A -85,B 0,C 180,E1 22103.484,E2 22103.484} C_VEL
LIN {X 0,Y 457.078,Z 373.772,A -85,B 0,C 180,E1 22099.811,E2 22099.811} C_VEL
LIN {X 0,Y 457.066,Z 373.765,A -85,B 0,C 180,E1 22096.095,E2 22096.095} C_VEL
LIN {X 0,Y 457.042,Z 373.785,A -85,B 0,C 180,E1 22092.502,E2 22092.502} C_VEL
LIN {X 0,Y 457.089,Z 374.053,A -85,B 0,C 180,E1 22091.07,E2 22091.07} C_VEL
LIN {X 0,Y 458.466,Z 377.431,A -85,B 0,C 180,E1 22090.436,E2 22090.436} C_VEL
LIN {X 0,Y 464.489,Z 391.058,A -85,B 0,C 180,E1 22088.161,E2 22088.161} C_VEL
LIN {X 0,Y 476.659,Z 410.235,A -85,B 0,C 180,E1 22086.519,E2 22086.519} C_VEL
LIN {X 0,Y 480.444,Z 416.884,A -85,B 0,C 180,E1 22086.023,E2 22086.023} C_VEL
LIN {X 0,Y 478.48,Z 523.503,A -85,B 0,C 180,E1 22084.324,E2 22084.324} C_VEL
LIN {X 0,Y 477.584,Z 531.203,A -85,B 0,C 180,E1 22084.274,E2 22084.274} C_VEL
LIN {X 0,Y 472.262,Z 551.748,A -85,B 0,C 180,E1 22084.412,E2 22084.412} C_VEL
LIN {X 0,Y 471.545,Z 558.359,A -85,B 0,C 180,E1 22084.363,E2 22084.363} C_VEL
LIN {X 0,Y 469.858,Z 654.174,A -85,B 0,C 180,E1 22082.811,E2 22082.811} C_VEL
LIN {X 0,Y 469.065,Z 674.364,A -85,B 0,C 180,E1 22082.261,E2 22082.261} C_VEL
LIN {X 0,Y 467.923,Z 693.41,A -85,B 0,C 180,E1 22081.528,E2 22081.528} C_VEL
LIN {X 0,Y 466.425,Z 711.957,A -85,B 0,C 180,E1 22080.601,E2 22080.601} C_VEL
LIN {X 0,Y 464.628,Z 730.236,A -85,B 0,C 180,E1 22079.45,E2 22079.45} C_VEL
LIN {X 0,Y 462.57,Z 747.452,A -85,B 0,C 180,E1 22078.11,E2 22078.11} C_VEL
LIN {X 0,Y 460.382,Z 763.822,A -85,B 0,C 180,E1 22076.573,E2 22076.573} C_VEL
LIN {X 0,Y 458.065,Z 779.874,A -85,B 0,C 180,E1 22074.764,E2 22074.764} C_VEL
LIN {X 0,Y 455.927,Z 794.121,A -85,B 0,C 180,E1 22072.837,E2 22072.837} C_VEL
LIN {X 0,Y 453.95,Z 807.007,A -85,B 0,C 180,E1 22070.767,E2 22070.767} C_VEL
LIN {X 0,Y 452.167,Z 819.108,A -85,B 0,C 180,E1 22068.431,E2 22068.431} C_VEL
LIN {X 0,Y 450.699,Z 829.667,A -85,B 0,C 180,E1 22065.965,E2 22065.965} C_VEL
LIN {X 0,Y 449.683,Z 838.284,A -85,B 0,C 180,E1 22063.499,E2 22063.499} C_VEL
LIN {X 0,Y 448.94,Z 845.572,A -85,B 0,C 180,E1 22060.911,E2 22060.911} C_VEL
LIN {X 0,Y 448.52,Z 851.397,A -85,B 0,C 180,E1 22058.196,E2 22058.196} C_VEL
LIN {X 0,Y 448.278,Z 855.485,A -85,B 0,C 180,E1 22055.503,E2 22055.503} C_VEL
LIN {X 0,Y 448.187,Z 857.964,A -85,B 0,C 180,E1 22052.812,E2 22052.812} C_VEL
LIN {X 0,Y 448.167,Z 858.852,A -85,B 0,C 180,E1 22050,E2 22050} C_VEL
LIN {X 0,Y 448.178,Z 858.069,A -85,B 0,C 180,E1 22047.315,E2 22047.315} C_VEL
LIN {X 0,Y 448.267,Z 855.733,A -85,B 0,C 180,E1 22044.625,E2 22044.625} C_VEL
LIN {X 0,Y 448.501,Z 851.777,A -85,B 0,C 180,E1 22041.927,E2 22041.927} C_VEL
LIN {X 0,Y 448.905,Z 846.049,A -85,B 0,C 180,E1 22039.191,E2 22039.191} C_VEL
LIN {X 0,Y 449.619,Z 838.989,A -85,B 0,C 180,E1 22036.629,E2 22036.629} C_VEL
LIN {X 0,Y 450.661,Z 830.018,A -85,B 0,C 180,E1 22034.032,E2 22034.032} C_VEL
LIN {X 0,Y 452.113,Z 819.531,A -85,B 0,C 180,E1 22031.565,E2 22031.565} C_VEL
LIN {X 0,Y 453.874,Z 807.479,A -85,B 0,C 180,E1 22029.228,E2 22029.228} C_VEL
LIN {X 0,Y 455.838,Z 794.685,A -85,B 0,C 180,E1 22027.157,E2 22027.157} C_VEL
LIN {X 0,Y 457.976,Z 780.473,A -85,B 0,C 180,E1 22025.22,E2 22025.22} C_VEL
LIN {X 0,Y 460.281,Z 764.636,A -85,B 0,C 180,E1 22023.42,E2 22023.42} C_VEL
LIN {X 0,Y 462.458,Z 748.44,A -85,B 0,C 180,E1 22021.882,E2 22021.882} C_VEL
LIN {X 0,Y 464.501,Z 731.348,A -85,B 0,C 180,E1 22020.54,E2 22020.54} C_VEL
LIN {X 0,Y 466.292,Z 713.346,A -85,B 0,C 180,E1 22019.388,E2 22019.388} C_VEL
LIN {X 0,Y 467.852,Z 694.494,A -85,B 0,C 180,E1 22018.429,E2 22018.429} C_VEL
LIN {X 0,Y 469.034,Z 675.266,A -85,B 0,C 180,E1 22017.677,E2 22017.677} C_VEL
LIN {X 0,Y 469.851,Z 654.886,A -85,B 0,C 180,E1 22017.112,E2 22017.112} C_VEL
LIN {X 0,Y 471.031,Z 588.357,A -85,B 0,C 180,E1 22016.021,E2 22016.021} C_VEL
LIN {X 0,Y 474.177,Z 419.609,A -85,B 0,C 180,E1 22013.308,E2 22013.308} C_VEL
LIN {X 0,Y 461.669,Z 399.545,A -85,B 0,C 180,E1 22011.604,E2 22011.604} C_VEL
LIN {X 0,Y 456.223,Z 391.121,A -85,B 0,C 180,E1 22010.781,E2 22010.781} C_VEL
LIN {X 0,Y 450.684,Z 378.586,A -85,B 0,C 180,E1 22008.579,E2 22008.579} C_VEL
LIN {X 0,Y 449.17,Z 375.071,A -85,B 0,C 180,E1 22007.892,E2 22007.892} C_VEL
LIN {X 0,Y 449.133,Z 374.792,A -85,B 0,C 180,E1 22006.531,E2 22006.531} C_VEL
LIN {X 0,Y 449.105,Z 374.768,A -85,B 0,C 180,E1 22002.912,E2 22002.912} C_VEL
LIN {X 0,Y 449.097,Z 374.75,A -85,B 0,C 180,E1 21999.22,E2 21999.22} C_VEL
LIN {X 0,Y 449.124,Z 374.793,A -85,B 0,C 180,E1 21995.525,E2 21995.525} C_VEL
LIN {X 0,Y 449.139,Z 374.786,A -85,B 0,C 180,E1 21991.754,E2 21991.754} C_VEL
LIN {X 0,Y 449.127,Z 374.787,A -85,B 0,C 180,E1 21988.017,E2 21988.017} C_VEL
LIN {X 0,Y 449.095,Z 374.79,A -85,B 0,C 180,E1 21984.323,E2 21984.323} C_VEL
LIN {X 0,Y 449.088,Z 374.79,A -85,B 0,C 180,E1 21980.596,E2 21980.596} C_VEL
LIN {X 0,Y 449.108,Z 374.793,A -85,B 0,C 180,E1 21976.957,E2 21976.957} C_VEL
LIN {X 0,Y 449.135,Z 374.786,A -85,B 0,C 180,E1 21973.256,E2 21973.256} C_VEL
LIN {X 0,Y 449.106,Z 374.782,A -85,B 0,C 180,E1 21969.539,E2 21969.539} C_VEL
LIN {X 0,Y 449.073,Z 374.778,A -85,B 0,C 180,E1 21966.007,E2 21966.007} C_VEL
LIN {X 0,Y 449.078,Z 374.782,A -85,B 0,C 180,E1 21962.297,E2 21962.297} C_VEL
LIN {X 0,Y 449.118,Z 374.788,A -85,B 0,C 180,E1 21958.725,E2 21958.725} C_VEL
LIN {X 0,Y 449.105,Z 374.793,A -85,B 0,C 180,E1 21955.019,E2 21955.019} C_VEL
LIN {X 0,Y 449.062,Z 374.794,A -85,B 0,C 180,E1 21951.55,E2 21951.55} C_VEL
LIN {X 0,Y 449.062,Z 374.794,A -85,B 0,C 180,E1 21947.786,E2 21947.786} C_VEL
LIN {X 0,Y 449.096,Z 374.785,A -85,B 0,C 180,E1 21944.24,E2 21944.24} C_VEL
LIN {X 0,Y 449.104,Z 374.783,A -85,B 0,C 180,E1 21940.492,E2 21940.492} C_VEL
LIN {X 0,Y 449.061,Z 374.761,A -85,B 0,C 180,E1 21936.929,E2 21936.929} C_VEL
LIN {X 0,Y 449.062,Z 374.798,A -85,B 0,C 180,E1 21933.223,E2 21933.223} C_VEL
LIN {X 0,Y 449.084,Z 374.752,A -85,B 0,C 180,E1 21929.642,E2 21929.642} C_VEL
LIN {X 0,Y 449.12,Z 374.776,A -85,B 0,C 180,E1 21926.028,E2 21926.028} C_VEL
LIN {X 0,Y 449.084,Z 374.787,A -85,B 0,C 180,E1 21922.408,E2 21922.408} C_VEL
LIN {X 0,Y 449.164,Z 375.118,A -85,B 0,C 180,E1 21921.606,E2 21921.606} C_VEL
LIN {X 0,Y 450.436,Z 378.34,A -85,B 0,C 180,E1 21921.084,E2 21921.084} C_VEL
LIN {X 0,Y 451.697,Z 380.504,A -85,B 0,C 180,E1 21920.723,E2 21920.723} C_VEL
LIN {X 0,Y 458.297,Z 393.245,A -85,B 0,C 180,E1 21918.787,E2 21918.787} C_VEL
LIN {X 0,Y 466.929,Z 411.329,A -85,B 0,C 180,E1 21916.324,E2 21916.324} C_VEL
LIN {X 0,Y 474.131,Z 427.933,A -85,B 0,C 180,E1 21914.294,E2 21914.294} C_VEL
LIN {X 0,Y 472.685,Z 449.07,A -85,B 0,C 180,E1 21912.885,E2 21912.885} C_VEL
LIN {X 0,Y 476.713,Z 482.649,A -85,B 0,C 180,E1 21911.824,E2 21911.824} C_VEL
LIN {X 0,Y 471.37,Z 709.821,A -85,B 0,C 180,E1 21907.921,E2 21907.921} C_VEL
LIN {X 0,Y 470.193,Z 756.6,A -85,B 0,C 180,E1 21907.097,E2 21907.097} C_VEL
LIN {X 0,Y 468.882,Z 779.293,A -85,B 0,C 180,E1 21906.492,E2 21906.492} C_VEL
LIN {X 0,Y 467.328,Z 800.822,A -85,B 0,C 180,E1 21905.698,E2 21905.698} C_VEL
LIN {X 0,Y 465.513,Z 822.291,A -85,B 0,C 180,E1 21904.69,E2 21904.69} C_VEL
LIN {X 0,Y 463.528,Z 843.704,A -85,B 0,C 180,E1 21903.441,E2 21903.441} C_VEL
LIN {X 0,Y 461.405,Z 864.19,A -85,B 0,C 180,E1 21901.984,E2 21901.984} C_VEL
LIN {X 0,Y 459.291,Z 883.81,A -85,B 0,C 180,E1 21900.332,E2 21900.332} C_VEL
LIN {X 0,Y 457.249,Z 901.955,A -85,B 0,C 180,E1 21898.538,E2 21898.538} C_VEL
LIN {X 0,Y 455.343,Z 918.95,A -85,B 0,C 180,E1 21896.573,E2 21896.573} C_VEL
LIN {X 0,Y 453.568,Z 934.855,A -85,B 0,C 180,E1 21894.436,E2 21894.436} C_VEL
LIN {X 0,Y 452.052,Z 949.157,A -85,B 0,C 180,E1 21892.222,E2 21892.222} C_VEL
LIN {X 0,Y 450.94,Z 960.098,A -85,B 0,C 180,E1 21890.235,E2 21890.235} C_VEL
LIN {X 0,Y 449.917,Z 970.267,A -85,B 0,C 180,E1 21887.983,E2 21887.983} C_VEL
LIN {X 0,Y 449.039,Z 980.053,A -85,B 0,C 180,E1 21885.364,E2 21885.364} C_VEL
LIN {X 0,Y 448.445,Z 988.47,A -85,B 0,C 180,E1 21882.62,E2 21882.62} C_VEL
LIN {X 0,Y 448.125,Z 994.873,A -85,B 0,C 180,E1 21880.022,E2 21880.022} C_VEL
LIN {X 0,Y 447.964,Z 999.606,A -85,B 0,C 180,E1 21877.438,E2 21877.438} C_VEL
LIN {X 0,Y 447.913,Z 1003.104,A -85,B 0,C 180,E1 21874.738,E2 21874.738} C_VEL
LIN {X 0,Y 447.908,Z 1004.949,A -85,B 0,C 180,E1 21872.175,E2 21872.175} C_VEL
LIN {X 0,Y 447.894,Z 1005.394,A -85,B 0,C 180,E1 21869.361,E2 21869.361} C_VEL
LIN {X 0,Y 447.908,Z 1004.334,A -85,B 0,C 180,E1 21866.674,E2 21866.674} C_VEL
LIN {X 0,Y 447.944,Z 1001.617,A -85,B 0,C 180,E1 21863.979,E2 21863.979} C_VEL
LIN {X 0,Y 448.049,Z 997.163,A -85,B 0,C 180,E1 21861.144,E2 21861.144} C_VEL
LIN {X 0,Y 448.301,Z 991.253,A -85,B 0,C 180,E1 21858.422,E2 21858.422} C_VEL
LIN {X 0,Y 448.757,Z 983.662,A -85,B 0,C 180,E1 21855.743,E2 21855.743} C_VEL
LIN {X 0,Y 449.551,Z 973.841,A -85,B 0,C 180,E1 21852.93,E2 21852.93} C_VEL
LIN {X 0,Y 450.617,Z 963.356,A -85,B 0,C 180,E1 21850.427,E2 21850.427} C_VEL
LIN {X 0,Y 451.65,Z 952.985,A -85,B 0,C 180,E1 21848.442,E2 21848.442} C_VEL
LIN {X 0,Y 453.116,Z 939.159,A -85,B 0,C 180,E1 21846.186,E2 21846.186} C_VEL
LIN {X 0,Y 454.795,Z 923.83,A -85,B 0,C 180,E1 21844.05,E2 21844.05} C_VEL
LIN {X 0,Y 456.778,Z 906.178,A -85,B 0,C 180,E1 21841.929,E2 21841.929} C_VEL
LIN {X 0,Y 458.806,Z 888.135,A -85,B 0,C 180,E1 21840.067,E2 21840.067} C_VEL
LIN {X 0,Y 460.892,Z 869.223,A -85,B 0,C 180,E1 21838.409,E2 21838.409} C_VEL
LIN {X 0,Y 462.922,Z 849.261,A -85,B 0,C 180,E1 21836.933,E2 21836.933} C_VEL
LIN {X 0,Y 465.087,Z 827.119,A -85,B 0,C 180,E1 21835.574,E2 21835.574} C_VEL
LIN {X 0,Y 466.902,Z 806.31,A -85,B 0,C 180,E1 21834.53,E2 21834.53} C_VEL
LIN {X 0,Y 468.542,Z 784.409,A -85,B 0,C 180,E1 21833.677,E2 21833.677} C_VEL
LIN {X 0,Y 469.909,Z 761.859,A -85,B 0,C 180,E1 21833.028,E2 21833.028} C_VEL
LIN {X 0,Y 470.817,Z 736.096,A -85,B 0,C 180,E1 21832.522,E2 21832.522} C_VEL
LIN {X 0,Y 476.013,Z 511.007,A -85,B 0,C 180,E1 21828.662,E2 21828.662} C_VEL
LIN {X 0,Y 476.577,Z 480.105,A -85,B 0,C 180,E1 21828.112,E2 21828.112} C_VEL
LIN {X 0,Y 472.644,Z 447.688,A -85,B 0,C 180,E1 21827.05,E2 21827.05} C_VEL
LIN {X 0,Y 474.066,Z 427.784,A -85,B 0,C 180,E1 21825.69,E2 21825.69} C_VEL
LIN {X 0,Y 465.838,Z 409.045,A -85,B 0,C 180,E1 21823.38,E2 21823.38} C_VEL
LIN {X 0,Y 457.423,Z 391.613,A -85,B 0,C 180,E1 21820.976,E2 21820.976} C_VEL
LIN {X 0,Y 452.877,Z 382.83,A -85,B 0,C 180,E1 21819.646,E2 21819.646} C_VEL
LIN {X 0,Y 450.874,Z 378.915,A -85,B 0,C 180,E1 21819.035,E2 21819.035} C_VEL
LIN {X 0,Y 449.202,Z 375.371,A -85,B 0,C 180,E1 21818.471,E2 21818.471} C_VEL
LIN {X 0,Y 449.13,Z 374.793,A -85,B 0,C 180,E1 21818.209,E2 21818.209} C_VEL
LIN {X 0,Y 449.084,Z 374.767,A -85,B 0,C 180,E1 21814.544,E2 21814.544} C_VEL
LIN {X 0,Y 449.062,Z 374.757,A -85,B 0,C 180,E1 21810.953,E2 21810.953} C_VEL
LIN {X 0,Y 449.079,Z 374.797,A -85,B 0,C 180,E1 21807.3,E2 21807.3} C_VEL
LIN {X 0,Y 449.108,Z 374.747,A -85,B 0,C 180,E1 21803.624,E2 21803.624} C_VEL
LIN {X 0,Y 449.084,Z 374.793,A -85,B 0,C 180,E1 21800.04,E2 21800.04} C_VEL
LIN {X 0,Y 449.054,Z 374.797,A -85,B 0,C 180,E1 21796.426,E2 21796.426} C_VEL
LIN {X 0,Y 449.061,Z 374.795,A -85,B 0,C 180,E1 21792.734,E2 21792.734} C_VEL
LIN {X 0,Y 449.098,Z 374.794,A -85,B 0,C 180,E1 21789.095,E2 21789.095} C_VEL
LIN {X 0,Y 449.1,Z 374.79,A -85,B 0,C 180,E1 21785.493,E2 21785.493} C_VEL
LIN {X 0,Y 449.067,Z 374.787,A -85,B 0,C 180,E1 21781.914,E2 21781.914} C_VEL
LIN {X 0,Y 449.068,Z 374.78,A -85,B 0,C 180,E1 21778.213,E2 21778.213} C_VEL
LIN {X 0,Y 449.105,Z 374.777,A -85,B 0,C 180,E1 21774.634,E2 21774.634} C_VEL
LIN {X 0,Y 449.113,Z 374.788,A -85,B 0,C 180,E1 21771.034,E2 21771.034} C_VEL
LIN {X 0,Y 449.084,Z 374.793,A -85,B 0,C 180,E1 21767.397,E2 21767.397} C_VEL
LIN {X 0,Y 449.08,Z 374.792,A -85,B 0,C 180,E1 21763.708,E2 21763.708} C_VEL
LIN {X 0,Y 449.106,Z 374.785,A -85,B 0,C 180,E1 21760.085,E2 21760.085} C_VEL
LIN {X 0,Y 449.133,Z 374.778,A -85,B 0,C 180,E1 21756.505,E2 21756.505} C_VEL
LIN {X 0,Y 449.102,Z 374.781,A -85,B 0,C 180,E1 21752.845,E2 21752.845} C_VEL
LIN {X 0,Y 449.091,Z 374.781,A -85,B 0,C 180,E1 21749.198,E2 21749.198} C_VEL
LIN {X 0,Y 449.11,Z 374.783,A -85,B 0,C 180,E1 21745.564,E2 21745.564} C_VEL
LIN {X 0,Y 449.135,Z 374.747,A -85,B 0,C 180,E1 21741.928,E2 21741.928} C_VEL
LIN {X 0,Y 449.128,Z 374.792,A -85,B 0,C 180,E1 21738.219,E2 21738.219} C_VEL
LIN {X 0,Y 449.102,Z 374.766,A -85,B 0,C 180,E1 21734.525,E2 21734.525} C_VEL
LIN {X 0,Y 449.165,Z 375.04,A -85,B 0,C 180,E1 21732.019,E2 21732.019} C_VEL
LIN {X 0,Y 450.465,Z 378.275,A -85,B 0,C 180,E1 21731.389,E2 21731.389} C_VEL
LIN {X 0,Y 456.487,Z 391.695,A -85,B 0,C 180,E1 21729.048,E2 21729.048} C_VEL
LIN {X 0,Y 469.465,Z 411.894,A -85,B 0,C 180,E1 21727.224,E2 21727.224} C_VEL
LIN {X 0,Y 474.204,Z 419.999,A -85,B 0,C 180,E1 21726.586,E2 21726.586} C_VEL
LIN {X 0,Y 471.545,Z 558.359,A -85,B 0,C 180,E1 21724.363,E2 21724.363} C_VEL
LIN {X 0,Y 470.614,Z 566.061,A -85,B 0,C 180,E1 21724.316,E2 21724.316} C_VEL
LIN {X 0,Y 465.276,Z 586.601,A -85,B 0,C 180,E1 21724.459,E2 21724.459} C_VEL
LIN {X 0,Y 464.576,Z 593.209,A -85,B 0,C 180,E1 21724.408,E2 21724.408} C_VEL
LIN {X 0,Y 463.398,Z 655.897,A -85,B 0,C 180,E1 21723.368,E2 21723.368} C_VEL
LIN {X 0,Y 462.55,Z 676.374,A -85,B 0,C 180,E1 21722.793,E2 21722.793} C_VEL
LIN {X 0,Y 461.315,Z 695.585,A -85,B 0,C 180,E1 21722.033,E2 21722.033} C_VEL
LIN {X 0,Y 459.63,Z 715.007,A -85,B 0,C 180,E1 21721.031,E2 21721.031} C_VEL
LIN {X 0,Y 457.747,Z 732.932,A -85,B 0,C 180,E1 21719.865,E2 21719.865} C_VEL
LIN {X 0,Y 455.611,Z 750.01,A -85,B 0,C 180,E1 21718.506,E2 21718.506} C_VEL
LIN {X 0,Y 453.322,Z 766.172,A -85,B 0,C 180,E1 21716.949,E2 21716.949} C_VEL
LIN {X 0,Y 450.984,Z 781.481,A -85,B 0,C 180,E1 21715.19,E2 21715.19} C_VEL
LIN {X 0,Y 448.715,Z 795.811,A -85,B 0,C 180,E1 21713.226,E2 21713.226} C_VEL
LIN {X 0,Y 446.626,Z 808.706,A -85,B 0,C 180,E1 21711.124,E2 21711.124} C_VEL
LIN {X 0,Y 444.718,Z 820.781,A -85,B 0,C 180,E1 21708.752,E2 21708.752} C_VEL
LIN {X 0,Y 443.125,Z 831.254,A -85,B 0,C 180,E1 21706.246,E2 21706.246} C_VEL
LIN {X 0,Y 442.006,Z 839.805,A -85,B 0,C 180,E1 21703.738,E2 21703.738} C_VEL
LIN {X 0,Y 441.174,Z 847.062,A -85,B 0,C 180,E1 21701.086,E2 21701.086} C_VEL
LIN {X 0,Y 440.693,Z 852.773,A -85,B 0,C 180,E1 21698.348,E2 21698.348} C_VEL
LIN {X 0,Y 440.43,Z 856.693,A -85,B 0,C 180,E1 21695.732,E2 21695.732} C_VEL
LIN {X 0,Y 440.309,Z 859.228,A -85,B 0,C 180,E1 21692.993,E2 21692.993} C_VEL
LIN {X 0,Y 440.271,Z 860.138,A -85,B 0,C 180,E1 21690.26,E2 21690.26} C_VEL
LIN {X 0,Y 440.29,Z 859.521,A -85,B 0,C 180,E1 21687.527,E2 21687.527} C_VEL
LIN {X 0,Y 440.392,Z 857.365,A -85,B 0,C 180,E1 21684.79,E2 21684.79} C_VEL
LIN {X 0,Y 440.639,Z 853.614,A -85,B 0,C 180,E1 21682.044,E2 21682.044} C_VEL
LIN {X 0,Y 441.054,Z 848.503,A -85,B 0,C 180,E1 21679.42,E2 21679.42} C_VEL
LIN {X 0,Y 441.844,Z 841.315,A -85,B 0,C 180,E1 21676.656,E2 21676.656} C_VEL
LIN {X 0,Y 442.945,Z 832.569,A -85,B 0,C 180,E1 21674.016,E2 21674.016} C_VEL
LIN {X 0,Y 444.464,Z 822.33,A -85,B 0,C 180,E1 21671.508,E2 21671.508} C_VEL
LIN {X 0,Y 446.187,Z 811.294,A -85,B 0,C 180,E1 21669.266,E2 21669.266} C_VEL
LIN {X 0,Y 448.343,Z 798.088,A -85,B 0,C 180,E1 21667.031,E2 21667.031} C_VEL
LIN {X 0,Y 450.566,Z 784.228,A -85,B 0,C 180,E1 21665.065,E2 21665.065} C_VEL
LIN {X 0,Y 452.971,Z 768.861,A -85,B 0,C 180,E1 21663.24,E2 21663.24} C_VEL
LIN {X 0,Y 455.287,Z 752.372,A -85,B 0,C 180,E1 21661.614,E2 21661.614} C_VEL
LIN {X 0,Y 457.401,Z 735.741,A -85,B 0,C 180,E1 21660.253,E2 21660.253} C_VEL
LIN {X 0,Y 459.432,Z 717.12,A -85,B 0,C 180,E1 21659.003,E2 21659.003} C_VEL
LIN {X 0,Y 461.085,Z 698.826,A -85,B 0,C 180,E1 21658.021,E2 21658.021} C_VEL
LIN {X 0,Y 462.43,Z 679.141,A -85,B 0,C 180,E1 21657.209,E2 21657.209} C_VEL
LIN {X 0,Y 463.289,Z 658.869,A -85,B 0,C 180,E1 21656.613,E2 21656.613} C_VEL
LIN {X 0,Y 463.882,Z 631.022,A -85,B 0,C 180,E1 21656.104,E2 21656.104} C_VEL
LIN {X 0,Y 468.041,Z 422.891,A -85,B 0,C 180,E1 21652.737,E2 21652.737} C_VEL
LIN {X 0,Y 455.469,Z 402.763,A -85,B 0,C 180,E1 21650.97,E2 21650.97} C_VEL
LIN {X 0,Y 448.407,Z 392.023,A -85,B 0,C 180,E1 21649.883,E2 21649.883} C_VEL
LIN {X 0,Y 442.739,Z 379.604,A -85,B 0,C 180,E1 21647.602,E2 21647.602} C_VEL
LIN {X 0,Y 441.208,Z 375.997,A -85,B 0,C 180,E1 21646.863,E2 21646.863} C_VEL
LIN {X 0,Y 441.163,Z 375.749,A -85,B 0,C 180,E1 21643.193,E2 21643.193} C_VEL
LIN {X 0,Y 441.177,Z 375.739,A -85,B 0,C 180,E1 21639.557,E2 21639.557} C_VEL
LIN {X 0,Y 441.197,Z 375.78,A -85,B 0,C 180,E1 21635.781,E2 21635.781} C_VEL
LIN {X 0,Y 441.196,Z 375.78,A -85,B 0,C 180,E1 21632.026,E2 21632.026} C_VEL
LIN {X 0,Y 441.161,Z 375.781,A -85,B 0,C 180,E1 21628.422,E2 21628.422} C_VEL
LIN {X 0,Y 441.152,Z 375.78,A -85,B 0,C 180,E1 21624.648,E2 21624.648} C_VEL
LIN {X 0,Y 441.165,Z 375.78,A -85,B 0,C 180,E1 21620.983,E2 21620.983} C_VEL
LIN {X 0,Y 441.193,Z 375.777,A -85,B 0,C 180,E1 21617.271,E2 21617.271} C_VEL
LIN {X 0,Y 441.187,Z 375.773,A -85,B 0,C 180,E1 21613.499,E2 21613.499} C_VEL
LIN {X 0,Y 441.149,Z 375.771,A -85,B 0,C 180,E1 21609.787,E2 21609.787} C_VEL
LIN {X 0,Y 441.134,Z 375.767,A -85,B 0,C 180,E1 21606.116,E2 21606.116} C_VEL
LIN {X 0,Y 441.148,Z 375.771,A -85,B 0,C 180,E1 21602.468,E2 21602.468} C_VEL
LIN {X 0,Y 441.188,Z 375.777,A -85,B 0,C 180,E1 21598.832,E2 21598.832} C_VEL
LIN {X 0,Y 441.162,Z 375.782,A -85,B 0,C 180,E1 21595.06,E2 21595.06} C_VEL
LIN {X 0,Y 441.124,Z 375.783,A -85,B 0,C 180,E1 21591.528,E2 21591.528} C_VEL
LIN {X 0,Y 441.121,Z 375.783,A -85,B 0,C 180,E1 21587.698,E2 21587.698} C_VEL
LIN {X 0,Y 441.143,Z 375.776,A -85,B 0,C 180,E1 21584.083,E2 21584.083} C_VEL
LIN {X 0,Y 441.169,Z 375.772,A -85,B 0,C 180,E1 21580.402,E2 21580.402} C_VEL
LIN {X 0,Y 441.131,Z 375.744,A -85,B 0,C 180,E1 21576.773,E2 21576.773} C_VEL
LIN {X 0,Y 441.123,Z 375.787,A -85,B 0,C 180,E1 21573.189,E2 21573.189} C_VEL
LIN {X 0,Y 441.144,Z 375.739,A -85,B 0,C 180,E1 21569.64,E2 21569.64} C_VEL
LIN {X 0,Y 441.18,Z 375.761,A -85,B 0,C 180,E1 21565.96,E2 21565.96} C_VEL
LIN {X 0,Y 441.157,Z 375.949,A -85,B 0,C 180,E1 21562.698,E2 21562.698} C_VEL
LIN {X 0,Y 441.73,Z 377.927,A -85,B 0,C 180,E1 21562.328,E2 21562.328} C_VEL
LIN {X 0,Y 443.78,Z 381.419,A -85,B 0,C 180,E1 21561.714,E2 21561.714} C_VEL
LIN {X 0,Y 450.244,Z 393.801,A -85,B 0,C 180,E1 21559.743,E2 21559.743} C_VEL
LIN {X 0,Y 459.16,Z 412.215,A -85,B 0,C 180,E1 21557.118,E2 21557.118} C_VEL
LIN {X 0,Y 467.474,Z 431.236,A -85,B 0,C 180,E1 21554.714,E2 21554.714} C_VEL
LIN {X 0,Y 466.269,Z 448.558,A -85,B 0,C 180,E1 21553.548,E2 21553.548} C_VEL
LIN {X 0,Y 470.43,Z 483.939,A -85,B 0,C 180,E1 21552.41,E2 21552.41} C_VEL
LIN {X 0,Y 464.727,Z 709.681,A -85,B 0,C 180,E1 21548.472,E2 21548.472} C_VEL
LIN {X 0,Y 463.463,Z 755.264,A -85,B 0,C 180,E1 21547.647,E2 21547.647} C_VEL
LIN {X 0,Y 462.033,Z 777.966,A -85,B 0,C 180,E1 21547.032,E2 21547.032} C_VEL
LIN {X 0,Y 460.397,Z 799.08,A -85,B 0,C 180,E1 21546.242,E2 21546.242} C_VEL
LIN {X 0,Y 458.448,Z 820.907,A -85,B 0,C 180,E1 21545.207,E2 21545.207} C_VEL
LIN {X 0,Y 456.363,Z 842.018,A -85,B 0,C 180,E1 21543.962,E2 21543.962} C_VEL
LIN {X 0,Y 454.16,Z 862.096,A -85,B 0,C 180,E1 21542.521,E2 21542.521} C_VEL
LIN {X 0,Y 451.872,Z 882.151,A -85,B 0,C 180,E1 21540.818,E2 21540.818} C_VEL
LIN {X 0,Y 449.727,Z 900.526,A -85,B 0,C 180,E1 21538.988,E2 21538.988} C_VEL
LIN {X 0,Y 447.81,Z 916.755,A -85,B 0,C 180,E1 21537.094,E2 21537.094} C_VEL
LIN {X 0,Y 445.915,Z 932.754,A -85,B 0,C 180,E1 21534.93,E2 21534.93} C_VEL
LIN {X 0,Y 444.281,Z 947.453,A -85,B 0,C 180,E1 21532.632,E2 21532.632} C_VEL
LIN {X 0,Y 442.908,Z 960.647,A -85,B 0,C 180,E1 21530.204,E2 21530.204} C_VEL
LIN {X 0,Y 441.791,Z 972.445,A -85,B 0,C 180,E1 21527.653,E2 21527.653} C_VEL
LIN {X 0,Y 441.187,Z 979.589,A -85,B 0,C 180,E1 21525.779,E2 21525.779} C_VEL
LIN {X 0,Y 440.53,Z 988.116,A -85,B 0,C 180,E1 21522.984,E2 21522.984} C_VEL
LIN {X 0,Y 440.17,Z 994.584,A -85,B 0,C 180,E1 21520.337,E2 21520.337} C_VEL
LIN {X 0,Y 439.981,Z 999.399,A -85,B 0,C 180,E1 21517.705,E2 21517.705} C_VEL
LIN {X 0,Y 439.91,Z 1002.876,A -85,B 0,C 180,E1 21515.085,E2 21515.085} C_VEL
LIN {X 0,Y 439.9,Z 1004.813,A -85,B 0,C 180,E1 21512.475,E2 21512.475} C_VEL
LIN {X 0,Y 439.9,Z 1005.462,A -85,B 0,C 180,E1 21509.74,E2 21509.74} C_VEL
LIN {X 0,Y 439.896,Z 1004.607,A -85,B 0,C 180,E1 21507.134,E2 21507.134} C_VEL
LIN {X 0,Y 439.935,Z 1002.096,A -85,B 0,C 180,E1 21504.262,E2 21504.262} C_VEL
LIN {X 0,Y 440.042,Z 998.158,A -85,B 0,C 180,E1 21501.508,E2 21501.508} C_VEL
LIN {X 0,Y 440.271,Z 992.465,A -85,B 0,C 180,E1 21498.739,E2 21498.739} C_VEL
LIN {X 0,Y 440.767,Z 984.694,A -85,B 0,C 180,E1 21495.821,E2 21495.821} C_VEL
LIN {X 0,Y 441.432,Z 976.76,A -85,B 0,C 180,E1 21493.42,E2 21493.42} C_VEL
LIN {X 0,Y 442.332,Z 966.49,A -85,B 0,C 180,E1 21491.007,E2 21491.007} C_VEL
LIN {X 0,Y 443.551,Z 954.352,A -85,B 0,C 180,E1 21488.584,E2 21488.584} C_VEL
LIN {X 0,Y 445.019,Z 940.811,A -85,B 0,C 180,E1 21486.289,E2 21486.289} C_VEL
LIN {X 0,Y 446.882,Z 924.56,A -85,B 0,C 180,E1 21483.922,E2 21483.922} C_VEL
LIN {X 0,Y 448.872,Z 907.794,A -85,B 0,C 180,E1 21481.825,E2 21481.825} C_VEL
LIN {X 0,Y 450.95,Z 890.07,A -85,B 0,C 180,E1 21479.931,E2 21479.931} C_VEL
LIN {X 0,Y 453.195,Z 870.794,A -85,B 0,C 180,E1 21478.181,E2 21478.181} C_VEL
LIN {X 0,Y 455.487,Z 849.82,A -85,B 0,C 180,E1 21476.57,E2 21476.57} C_VEL
LIN {X 0,Y 457.689,Z 829.02,A -85,B 0,C 180,E1 21475.242,E2 21475.242} C_VEL
LIN {X 0,Y 459.69,Z 807.418,A -85,B 0,C 180,E1 21474.12,E2 21474.12} C_VEL
LIN {X 0,Y 461.479,Z 785.557,A -85,B 0,C 180,E1 21473.23,E2 21473.23} C_VEL
LIN {X 0,Y 463.05,Z 762.471,A -85,B 0,C 180,E1 21472.528,E2 21472.528} C_VEL
LIN {X 0,Y 464.037,Z 739.151,A -85,B 0,C 180,E1 21472.037,E2 21472.037} C_VEL
LIN {X 0,Y 469.763,Z 509.187,A -85,B 0,C 180,E1 21468.029,E2 21468.029} C_VEL
LIN {X 0,Y 470.293,Z 481.426,A -85,B 0,C 180,E1 21467.527,E2 21467.527} C_VEL
LIN {X 0,Y 466.192,Z 447.532,A -85,B 0,C 180,E1 21466.412,E2 21466.412} C_VEL
LIN {X 0,Y 467.36,Z 430.951,A -85,B 0,C 180,E1 21465.257,E2 21465.257} C_VEL
LIN {X 0,Y 458.517,Z 410.834,A -85,B 0,C 180,E1 21462.701,E2 21462.701} C_VEL
LIN {X 0,Y 449.737,Z 392.857,A -85,B 0,C 180,E1 21460.12,E2 21460.12} C_VEL
LIN {X 0,Y 444.899,Z 383.759,A -85,B 0,C 180,E1 21458.665,E2 21458.665} C_VEL
LIN {X 0,Y 442.96,Z 379.893,A -85,B 0,C 180,E1 21458.04,E2 21458.04} C_VEL
LIN {X 0,Y 441.269,Z 376.516,A -85,B 0,C 180,E1 21457.473,E2 21457.473} C_VEL
LIN {X 0,Y 441.138,Z 375.812,A -85,B 0,C 180,E1 21457.24,E2 21457.24} C_VEL
LIN {X 0,Y 441.151,Z 375.778,A -85,B 0,C 180,E1 21453.574,E2 21453.574} C_VEL
LIN {X 0,Y 441.188,Z 375.735,A -85,B 0,C 180,E1 21449.906,E2 21449.906} C_VEL
LIN {X 0,Y 441.137,Z 375.77,A -85,B 0,C 180,E1 21446.375,E2 21446.375} C_VEL
LIN {X 0,Y 441.12,Z 375.756,A -85,B 0,C 180,E1 21442.664,E2 21442.664} C_VEL
LIN {X 0,Y 441.124,Z 375.774,A -85,B 0,C 180,E1 21438.912,E2 21438.912} C_VEL
LIN {X 0,Y 441.152,Z 375.771,A -85,B 0,C 180,E1 21435.243,E2 21435.243} C_VEL
LIN {X 0,Y 441.156,Z 375.771,A -85,B 0,C 180,E1 21431.637,E2 21431.637} C_VEL
LIN {X 0,Y 441.122,Z 375.781,A -85,B 0,C 180,E1 21428.078,E2 21428.078} C_VEL
LIN {X 0,Y 441.125,Z 375.783,A -85,B 0,C 180,E1 21424.289,E2 21424.289} C_VEL
LIN {X 0,Y 441.15,Z 375.783,A -85,B 0,C 180,E1 21420.649,E2 21420.649} C_VEL
LIN {X 0,Y 441.18,Z 375.773,A -85,B 0,C 180,E1 21417.012,E2 21417.012} C_VEL
LIN {X 0,Y 441.15,Z 375.766,A -85,B 0,C 180,E1 21413.362,E2 21413.362} C_VEL
LIN {X 0,Y 441.136,Z 375.768,A -85,B 0,C 180,E1 21409.685,E2 21409.685} C_VEL
LIN {X 0,Y 441.143,Z 375.774,A -85,B 0,C 180,E1 21405.922,E2 21405.922} C_VEL
LIN {X 0,Y 441.181,Z 375.776,A -85,B 0,C 180,E1 21402.32,E2 21402.32} C_VEL
LIN {X 0,Y 441.194,Z 375.779,A -85,B 0,C 180,E1 21398.6,E2 21398.6} C_VEL
LIN {X 0,Y 441.161,Z 375.782,A -85,B 0,C 180,E1 21394.924,E2 21394.924} C_VEL
LIN {X 0,Y 441.153,Z 375.782,A -85,B 0,C 180,E1 21391.282,E2 21391.282} C_VEL
LIN {X 0,Y 441.173,Z 375.781,A -85,B 0,C 180,E1 21387.665,E2 21387.665} C_VEL
LIN {X 0,Y 441.196,Z 375.776,A -85,B 0,C 180,E1 21383.898,E2 21383.898} C_VEL
LIN {X 0,Y 441.195,Z 375.74,A -85,B 0,C 180,E1 21380.107,E2 21380.107} C_VEL
LIN {X 0,Y 441.167,Z 375.745,A -85,B 0,C 180,E1 21376.45,E2 21376.45} C_VEL
LIN {X 0,Y 441.194,Z 375.957,A -85,B 0,C 180,E1 21373.047,E2 21373.047} C_VEL
LIN {X 0,Y 442.514,Z 379.3,A -85,B 0,C 180,E1 21372.366,E2 21372.366} C_VEL
LIN {X 0,Y 448.445,Z 392.094,A -85,B 0,C 180,E1 21370.015,E2 21370.015} C_VEL
LIN {X 0,Y 461.42,Z 412.053,A -85,B 0,C 180,E1 21368.081,E2 21368.081} C_VEL
LIN {X 0,Y 468.007,Z 423.217,A -85,B 0,C 180,E1 21367.163,E2 21367.163} C_VEL
LIN {X 0,Y 464.576,Z 593.209,A -85,B 0,C 180,E1 21364.408,E2 21364.408} C_VEL
LIN {X 0,Y 463.673,Z 600.905,A -85,B 0,C 180,E1 21364.358,E2 21364.358} C_VEL
LIN {X 0,Y 458.332,Z 621.438,A -85,B 0,C 180,E1 21364.504,E2 21364.504} C_VEL
LIN {X 0,Y 457.566,Z 628.049,A -85,B 0,C 180,E1 21364.459,E2 21364.459} C_VEL
LIN {X 0,Y 456.91,Z 658.868,A -85,B 0,C 180,E1 21363.905,E2 21363.905} C_VEL
LIN {X 0,Y 456.019,Z 679.492,A -85,B 0,C 180,E1 21363.301,E2 21363.301} C_VEL
LIN {X 0,Y 454.68,Z 698.435,A -85,B 0,C 180,E1 21362.521,E2 21362.521} C_VEL
LIN {X 0,Y 452.969,Z 716.905,A -85,B 0,C 180,E1 21361.539,E2 21361.539} C_VEL
LIN {X 0,Y 450.88,Z 735.559,A -85,B 0,C 180,E1 21360.294,E2 21360.294} C_VEL
LIN {X 0,Y 448.656,Z 752.464,A -85,B 0,C 180,E1 21358.917,E2 21358.917} C_VEL
LIN {X 0,Y 446.179,Z 769.084,A -85,B 0,C 180,E1 21357.272,E2 21357.272} C_VEL
LIN {X 0,Y 443.721,Z 784.126,A -85,B 0,C 180,E1 21355.489,E2 21355.489} C_VEL
LIN {X 0,Y 441.349,Z 798.245,A -85,B 0,C 180,E1 21353.495,E2 21353.495} C_VEL
LIN {X 0,Y 439.156,Z 810.971,A -85,B 0,C 180,E1 21351.361,E2 21351.361} C_VEL
LIN {X 0,Y 437.258,Z 822.353,A -85,B 0,C 180,E1 21349.084,E2 21349.084} C_VEL
LIN {X 0,Y 435.558,Z 832.824,A -85,B 0,C 180,E1 21346.536,E2 21346.536} C_VEL
LIN {X 0,Y 434.335,Z 841.315,A -85,B 0,C 180,E1 21343.986,E2 21343.986} C_VEL
LIN {X 0,Y 433.422,Z 848.467,A -85,B 0,C 180,E1 21341.307,E2 21341.307} C_VEL
LIN {X 0,Y 432.873,Z 854.177,A -85,B 0,C 180,E1 21338.5,E2 21338.5} C_VEL
LIN {X 0,Y 432.558,Z 858.196,A -85,B 0,C 180,E1 21335.703,E2 21335.703} C_VEL
LIN {X 0,Y 432.422,Z 860.633,A -85,B 0,C 180,E1 21332.915,E2 21332.915} C_VEL
LIN {X 0,Y 432.391,Z 861.508,A -85,B 0,C 180,E1 21330,E2 21330} C_VEL
LIN {X 0,Y 432.41,Z 860.734,A -85,B 0,C 180,E1 21327.217,E2 21327.217} C_VEL
LIN {X 0,Y 432.529,Z 858.575,A -85,B 0,C 180,E1 21324.562,E2 21324.562} C_VEL
LIN {X 0,Y 432.83,Z 854.775,A -85,B 0,C 180,E1 21321.766,E2 21321.766} C_VEL
LIN {X 0,Y 433.31,Z 849.626,A -85,B 0,C 180,E1 21319.094,E2 21319.094} C_VEL
LIN {X 0,Y 434.212,Z 842.419,A -85,B 0,C 180,E1 21316.281,E2 21316.281} C_VEL
LIN {X 0,Y 435.44,Z 833.649,A -85,B 0,C 180,E1 21313.596,E2 21313.596} C_VEL
LIN {X 0,Y 437.092,Z 823.314,A -85,B 0,C 180,E1 21311.046,E2 21311.046} C_VEL
LIN {X 0,Y 438.951,Z 812.142,A -85,B 0,C 180,E1 21308.768,E2 21308.768} C_VEL
LIN {X 0,Y 441.258,Z 798.798,A -85,B 0,C 180,E1 21306.499,E2 21306.499} C_VEL
LIN {X 0,Y 443.62,Z 784.79,A -85,B 0,C 180,E1 21304.504,E2 21304.504} C_VEL
LIN {X 0,Y 446.077,Z 769.882,A -85,B 0,C 180,E1 21302.72,E2 21302.72} C_VEL
LIN {X 0,Y 448.528,Z 753.339,A -85,B 0,C 180,E1 21301.073,E2 21301.073} C_VEL
LIN {X 0,Y 450.748,Z 736.631,A -85,B 0,C 180,E1 21299.695,E2 21299.695} C_VEL
LIN {X 0,Y 452.842,Z 718.26,A -85,B 0,C 180,E1 21298.45,E2 21298.45} C_VEL
LIN {X 0,Y 454.61,Z 699.486,A -85,B 0,C 180,E1 21297.435,E2 21297.435} C_VEL
LIN {X 0,Y 456.004,Z 679.899,A -85,B 0,C 180,E1 21296.621,E2 21296.621} C_VEL
LIN {X 0,Y 456.9,Z 659.446,A -85,B 0,C 180,E1 21296.018,E2 21296.018} C_VEL
LIN {X 0,Y 457.537,Z 630.379,A -85,B 0,C 180,E1 21295.487,E2 21295.487} C_VEL
LIN {X 0,Y 461.813,Z 426.033,A -85,B 0,C 180,E1 21292.134,E2 21292.134} C_VEL
LIN {X 0,Y 449.424,Z 406.148,A -85,B 0,C 180,E1 21290.333,E2 21290.333} C_VEL
LIN {X 0,Y 440.476,Z 392.752,A -85,B 0,C 180,E1 21288.906,E2 21288.906} C_VEL
LIN {X 0,Y 436.185,Z 383.782,A -85,B 0,C 180,E1 21287.184,E2 21287.184} C_VEL
LIN {X 0,Y 434.484,Z 380.134,A -85,B 0,C 180,E1 21286.46,E2 21286.46} C_VEL
LIN {X 0,Y 433.279,Z 376.972,A -85,B 0,C 180,E1 21285.799,E2 21285.799} C_VEL
LIN {X 0,Y 433.259,Z 376.757,A -85,B 0,C 180,E1 21282.188,E2 21282.188} C_VEL
LIN {X 0,Y 433.234,Z 376.721,A -85,B 0,C 180,E1 21278.528,E2 21278.528} C_VEL
LIN {X 0,Y 433.221,Z 376.765,A -85,B 0,C 180,E1 21274.755,E2 21274.755} C_VEL
LIN {X 0,Y 433.219,Z 376.758,A -85,B 0,C 180,E1 21270.976,E2 21270.976} C_VEL
LIN {X 0,Y 433.245,Z 376.755,A -85,B 0,C 180,E1 21267.323,E2 21267.323} C_VEL
LIN {X 0,Y 433.259,Z 376.753,A -85,B 0,C 180,E1 21263.531,E2 21263.531} C_VEL
LIN {X 0,Y 433.237,Z 376.759,A -85,B 0,C 180,E1 21259.832,E2 21259.832} C_VEL
LIN {X 0,Y 433.208,Z 376.768,A -85,B 0,C 180,E1 21256.217,E2 21256.217} C_VEL
LIN {X 0,Y 433.205,Z 376.772,A -85,B 0,C 180,E1 21252.395,E2 21252.395} C_VEL
LIN {X 0,Y 433.226,Z 376.771,A -85,B 0,C 180,E1 21248.762,E2 21248.762} C_VEL
LIN {X 0,Y 433.246,Z 376.756,A -85,B 0,C 180,E1 21245.031,E2 21245.031} C_VEL
LIN {X 0,Y 433.231,Z 376.753,A -85,B 0,C 180,E1 21241.19,E2 21241.19} C_VEL
LIN {X 0,Y 433.192,Z 376.761,A -85,B 0,C 180,E1 21237.619,E2 21237.619} C_VEL
LIN {X 0,Y 433.189,Z 376.767,A -85,B 0,C 180,E1 21233.905,E2 21233.905} C_VEL
LIN {X 0,Y 433.213,Z 376.769,A -85,B 0,C 180,E1 21230.301,E2 21230.301} C_VEL
LIN {X 0,Y 433.238,Z 376.77,A -85,B 0,C 180,E1 21226.521,E2 21226.521} C_VEL
LIN {X 0,Y 433.202,Z 376.775,A -85,B 0,C 180,E1 21222.817,E2 21222.817} C_VEL
LIN {X 0,Y 433.179,Z 376.777,A -85,B 0,C 180,E1 21219.179,E2 21219.179} C_VEL
LIN {X 0,Y 433.178,Z 376.726,A -85,B 0,C 180,E1 21215.306,E2 21215.306} C_VEL
LIN {X 0,Y 433.203,Z 376.76,A -85,B 0,C 180,E1 21211.611,E2 21211.611} C_VEL
LIN {X 0,Y 433.239,Z 376.744,A -85,B 0,C 180,E1 21207.94,E2 21207.94} C_VEL
LIN {X 0,Y 433.227,Z 376.727,A -85,B 0,C 180,E1 21204.112,E2 21204.112} C_VEL
LIN {X 0,Y 433.304,Z 377.215,A -85,B 0,C 180,E1 21203.685,E2 21203.685} C_VEL
LIN {X 0,Y 434.703,Z 380.517,A -85,B 0,C 180,E1 21203.107,E2 21203.107} C_VEL
LIN {X 0,Y 435.916,Z 382.524,A -85,B 0,C 180,E1 21202.733,E2 21202.733} C_VEL
LIN {X 0,Y 443.038,Z 396.121,A -85,B 0,C 180,E1 21200.475,E2 21200.475} C_VEL
LIN {X 0,Y 451.226,Z 412.782,A -85,B 0,C 180,E1 21197.996,E2 21197.996} C_VEL
LIN {X 0,Y 459.511,Z 431.562,A -85,B 0,C 180,E1 21195.522,E2 21195.522} C_VEL
LIN {X 0,Y 460.842,Z 435.13,A -85,B 0,C 180,E1 21195.099,E2 21195.099} C_VEL
LIN {X 0,Y 459.886,Z 447.671,A -85,B 0,C 180,E1 21194.244,E2 21194.244} C_VEL
LIN {X 0,Y 464.193,Z 485.365,A -85,B 0,C 180,E1 21193.009,E2 21193.009} C_VEL
LIN {X 0,Y 458.16,Z 709.672,A -85,B 0,C 180,E1 21189.042,E2 21189.042} C_VEL
LIN {X 0,Y 456.837,Z 754.159,A -85,B 0,C 180,E1 21188.222,E2 21188.222} C_VEL
LIN {X 0,Y 455.31,Z 776.752,A -85,B 0,C 180,E1 21187.602,E2 21187.602} C_VEL
LIN {X 0,Y 453.481,Z 798.61,A -85,B 0,C 180,E1 21186.767,E2 21186.767} C_VEL
LIN {X 0,Y 451.34,Z 820.646,A -85,B 0,C 180,E1 21185.686,E2 21185.686} C_VEL
LIN {X 0,Y 449.126,Z 841.397,A -85,B 0,C 180,E1 21184.431,E2 21184.431} C_VEL
LIN {X 0,Y 446.757,Z 861.771,A -85,B 0,C 180,E1 21182.938,E2 21182.938} C_VEL
LIN {X 0,Y 444.388,Z 881.307,A -85,B 0,C 180,E1 21181.242,E2 21181.242} C_VEL
LIN {X 0,Y 442.15,Z 899.597,A -85,B 0,C 180,E1 21179.385,E2 21179.385} C_VEL
LIN {X 0,Y 439.99,Z 917.038,A -85,B 0,C 180,E1 21177.311,E2 21177.311} C_VEL
LIN {X 0,Y 438.037,Z 932.805,A -85,B 0,C 180,E1 21175.121,E2 21175.121} C_VEL
LIN {X 0,Y 436.263,Z 948.048,A -85,B 0,C 180,E1 21172.644,E2 21172.644} C_VEL
LIN {X 0,Y 434.875,Z 961.086,A -85,B 0,C 180,E1 21170.173,E2 21170.173} C_VEL
LIN {X 0,Y 433.758,Z 972.57,A -85,B 0,C 180,E1 21167.575,E2 21167.575} C_VEL
LIN {X 0,Y 432.919,Z 982.666,A -85,B 0,C 180,E1 21164.853,E2 21164.853} C_VEL
LIN {X 0,Y 432.454,Z 989.705,A -85,B 0,C 180,E1 21162.552,E2 21162.552} C_VEL
LIN {X 0,Y 432.134,Z 995.638,A -85,B 0,C 180,E1 21159.993,E2 21159.993} C_VEL
LIN {X 0,Y 431.967,Z 1000.225,A -85,B 0,C 180,E1 21157.314,E2 21157.314} C_VEL
LIN {X 0,Y 431.919,Z 1003.444,A -85,B 0,C 180,E1 21154.514,E2 21154.514} C_VEL
LIN {X 0,Y 431.901,Z 1005.209,A -85,B 0,C 180,E1 21151.725,E2 21151.725} C_VEL
LIN {X 0,Y 431.901,Z 1005.348,A -85,B 0,C 180,E1 21149.072,E2 21149.072} C_VEL
LIN {X 0,Y 431.913,Z 1004.123,A -85,B 0,C 180,E1 21146.284,E2 21146.284} C_VEL
LIN {X 0,Y 431.961,Z 1001.297,A -85,B 0,C 180,E1 21143.489,E2 21143.489} C_VEL
LIN {X 0,Y 432.091,Z 996.909,A -85,B 0,C 180,E1 21140.68,E2 21140.68} C_VEL
LIN {X 0,Y 432.34,Z 991.798,A -85,B 0,C 180,E1 21138.259,E2 21138.259} C_VEL
LIN {X 0,Y 432.791,Z 984.454,A -85,B 0,C 180,E1 21135.69,E2 21135.69} C_VEL
LIN {X 0,Y 433.528,Z 975.34,A -85,B 0,C 180,E1 21133.109,E2 21133.109} C_VEL
LIN {X 0,Y 434.546,Z 964.262,A -85,B 0,C 180,E1 21130.513,E2 21130.513} C_VEL
LIN {X 0,Y 435.922,Z 951.137,A -85,B 0,C 180,E1 21127.907,E2 21127.907} C_VEL
LIN {X 0,Y 437.62,Z 936.502,A -85,B 0,C 180,E1 21125.432,E2 21125.432} C_VEL
LIN {X 0,Y 439.517,Z 920.76,A -85,B 0,C 180,E1 21123.178,E2 21123.178} C_VEL
LIN {X 0,Y 441.671,Z 903.248,A -85,B 0,C 180,E1 21121.027,E2 21121.027} C_VEL
LIN {X 0,Y 443.97,Z 884.905,A -85,B 0,C 180,E1 21119.097,E2 21119.097} C_VEL
LIN {X 0,Y 446.373,Z 865.213,A -85,B 0,C 180,E1 21117.332,E2 21117.332} C_VEL
LIN {X 0,Y 448.67,Z 845.287,A -85,B 0,C 180,E1 21115.839,E2 21115.839} C_VEL
LIN {X 0,Y 450.991,Z 823.862,A -85,B 0,C 180,E1 21114.494,E2 21114.494} C_VEL
LIN {X 0,Y 453.154,Z 802.473,A -85,B 0,C 180,E1 21113.4,E2 21113.4} C_VEL
LIN {X 0,Y 454.96,Z 781.485,A -85,B 0,C 180,E1 21112.56,E2 21112.56} C_VEL
LIN {X 0,Y 456.53,Z 759.04,A -85,B 0,C 180,E1 21111.898,E2 21111.898} C_VEL
LIN {X 0,Y 457.587,Z 732.124,A -85,B 0,C 180,E1 21111.353,E2 21111.353} C_VEL
LIN {X 0,Y 463.794,Z 499.448,A -85,B 0,C 180,E1 21107.239,E2 21107.239} C_VEL
LIN {X 0,Y 464.068,Z 482.826,A -85,B 0,C 180,E1 21106.928,E2 21106.928} C_VEL
LIN {X 0,Y 459.842,Z 446.467,A -85,B 0,C 180,E1 21105.701,E2 21105.701} C_VEL
LIN {X 0,Y 460.76,Z 434.476,A -85,B 0,C 180,E1 21104.85,E2 21104.85} C_VEL
LIN {X 0,Y 452.04,Z 414.507,A -85,B 0,C 180,E1 21102.253,E2 21102.253} C_VEL
LIN {X 0,Y 443.817,Z 397.697,A -85,B 0,C 180,E1 21099.777,E2 21099.777} C_VEL
LIN {X 0,Y 437.448,Z 385.406,A -85,B 0,C 180,E1 21097.774,E2 21097.774} C_VEL
LIN {X 0,Y 435.117,Z 381.043,A -85,B 0,C 180,E1 21097.017,E2 21097.017} C_VEL
LIN {X 0,Y 433.369,Z 377.555,A -85,B 0,C 180,E1 21096.403,E2 21096.403} C_VEL
LIN {X 0,Y 433.243,Z 376.761,A -85,B 0,C 180,E1 21096.05,E2 21096.05} C_VEL
LIN {X 0,Y 433.229,Z 376.75,A -85,B 0,C 180,E1 21092.217,E2 21092.217} C_VEL
LIN {X 0,Y 433.187,Z 376.751,A -85,B 0,C 180,E1 21088.691,E2 21088.691} C_VEL
LIN {X 0,Y 433.18,Z 376.727,A -85,B 0,C 180,E1 21084.904,E2 21084.904} C_VEL
LIN {X 0,Y 433.2,Z 376.775,A -85,B 0,C 180,E1 21081.194,E2 21081.194} C_VEL
LIN {X 0,Y 433.227,Z 376.771,A -85,B 0,C 180,E1 21077.459,E2 21077.459} C_VEL
LIN {X 0,Y 433.218,Z 376.769,A -85,B 0,C 180,E1 21073.699,E2 21073.699} C_VEL
LIN {X 0,Y 433.19,Z 376.769,A -85,B 0,C 180,E1 21069.968,E2 21069.968} C_VEL
LIN {X 0,Y 433.182,Z 376.767,A -85,B 0,C 180,E1 21066.228,E2 21066.228} C_VEL
LIN {X 0,Y 433.196,Z 376.759,A -85,B 0,C 180,E1 21062.513,E2 21062.513} C_VEL
LIN {X 0,Y 433.241,Z 376.753,A -85,B 0,C 180,E1 21058.942,E2 21058.942} C_VEL
LIN {X 0,Y 433.236,Z 376.759,A -85,B 0,C 180,E1 21055.101,E2 21055.101} C_VEL
LIN {X 0,Y 433.202,Z 376.771,A -85,B 0,C 180,E1 21051.505,E2 21051.505} C_VEL
LIN {X 0,Y 433.2,Z 376.77,A -85,B 0,C 180,E1 21047.74,E2 21047.74} C_VEL
LIN {X 0,Y 433.216,Z 376.766,A -85,B 0,C 180,E1 21044.058,E2 21044.058} C_VEL
LIN {X 0,Y 433.253,Z 376.755,A -85,B 0,C 180,E1 21040.45,E2 21040.45} C_VEL
LIN {X 0,Y 433.24,Z 376.755,A -85,B 0,C 180,E1 21036.698,E2 21036.698} C_VEL
LIN {X 0,Y 433.218,Z 376.758,A -85,B 0,C 180,E1 21032.956,E2 21032.956} C_VEL
LIN {X 0,Y 433.213,Z 376.758,A -85,B 0,C 180,E1 21029.177,E2 21029.177} C_VEL
LIN {X 0,Y 433.223,Z 376.762,A -85,B 0,C 180,E1 21025.406,E2 21025.406} C_VEL
LIN {X 0,Y 433.247,Z 376.72,A -85,B 0,C 180,E1 21021.681,E2 21021.681} C_VEL
LIN {X 0,Y 433.261,Z 376.764,A -85,B 0,C 180,E1 21017.989,E2 21017.989} C_VEL
LIN {X 0,Y 433.248,Z 376.798,A -85,B 0,C 180,E1 21014.178,E2 21014.178} C_VEL
LIN {X 0,Y 433.621,Z 378.338,A -85,B 0,C 180,E1 21013.802,E2 21013.802} C_VEL
LIN {X 0,Y 435.653,Z 382.653,A -85,B 0,C 180,E1 21012.934,E2 21012.934} C_VEL
LIN {X 0,Y 439.234,Z 390.188,A -85,B 0,C 180,E1 21011.479,E2 21011.479} C_VEL
LIN {X 0,Y 441.107,Z 393.93,A -85,B 0,C 180,E1 21010.842,E2 21010.842} C_VEL
LIN {X 0,Y 454.459,Z 414.055,A -85,B 0,C 180,E1 21008.82,E2 21008.82} C_VEL
LIN {X 0,Y 461.859,Z 426.448,A -85,B 0,C 180,E1 21007.755,E2 21007.755} C_VEL
LIN {X 0,Y 457.566,Z 628.049,A -85,B 0,C 180,E1 21004.459,E2 21004.459} C_VEL
LIN {X 0,Y 456.599,Z 635.756,A -85,B 0,C 180,E1 21004.417,E2 21004.417} C_VEL
LIN {X 0,Y 451.205,Z 656.269,A -85,B 0,C 180,E1 21004.534,E2 21004.534} C_VEL
LIN {X 0,Y 450.481,Z 661.721,A -85,B 0,C 180,E1 21004.457,E2 21004.457} C_VEL
LIN {X 0,Y 450.433,Z 662.808,A -85,B 0,C 180,E1 21004.428,E2 21004.428} C_VEL
LIN {X 0,Y 449.456,Z 682.742,A -85,B 0,C 180,E1 21003.809,E2 21003.809} C_VEL
LIN {X 0,Y 448.018,Z 701.961,A -85,B 0,C 180,E1 21002.989,E2 21002.989} C_VEL
LIN {X 0,Y 446.119,Z 720.951,A -85,B 0,C 180,E1 21001.929,E2 21001.929} C_VEL
LIN {X 0,Y 443.927,Z 738.927,A -85,B 0,C 180,E1 21000.677,E2 21000.677} C_VEL
LIN {X 0,Y 441.479,Z 756.2,A -85,B 0,C 180,E1 20999.21,E2 20999.21} C_VEL
LIN {X 0,Y 438.934,Z 772.487,A -85,B 0,C 180,E1 20997.54,E2 20997.54} C_VEL
LIN {X 0,Y 436.212,Z 788.281,A -85,B 0,C 180,E1 20995.596,E2 20995.596} C_VEL
LIN {X 0,Y 433.678,Z 802.354,A -85,B 0,C 180,E1 20993.504,E2 20993.504} C_VEL
LIN {X 0,Y 431.373,Z 814.859,A -85,B 0,C 180,E1 20991.286,E2 20991.286} C_VEL
LIN {X 0,Y 429.371,Z 826.154,A -85,B 0,C 180,E1 20988.883,E2 20988.883} C_VEL
LIN {X 0,Y 427.658,Z 836.205,A -85,B 0,C 180,E1 20986.291,E2 20986.291} C_VEL
LIN {X 0,Y 426.443,Z 844.38,A -85,B 0,C 180,E1 20983.696,E2 20983.696} C_VEL
LIN {X 0,Y 425.491,Z 851.527,A -85,B 0,C 180,E1 20980.809,E2 20980.809} C_VEL
LIN {X 0,Y 424.945,Z 856.926,A -85,B 0,C 180,E1 20977.842,E2 20977.842} C_VEL
LIN {X 0,Y 424.646,Z 860.402,A -85,B 0,C 180,E1 20974.997,E2 20974.997} C_VEL
LIN {X 0,Y 424.521,Z 862.326,A -85,B 0,C 180,E1 20972.159,E2 20972.159} C_VEL
LIN {X 0,Y 424.495,Z 862.726,A -85,B 0,C 180,E1 20969.19,E2 20969.19} C_VEL
LIN {X 0,Y 424.566,Z 861.472,A -85,B 0,C 180,E1 20966.219,E2 20966.219} C_VEL
LIN {X 0,Y 424.791,Z 858.688,A -85,B 0,C 180,E1 20963.36,E2 20963.36} C_VEL
LIN {X 0,Y 425.19,Z 854.355,A -85,B 0,C 180,E1 20960.526,E2 20960.526} C_VEL
LIN {X 0,Y 425.945,Z 847.97,A -85,B 0,C 180,E1 20957.559,E2 20957.559} C_VEL
LIN {X 0,Y 427.056,Z 840.161,A -85,B 0,C 180,E1 20954.799,E2 20954.799} C_VEL
LIN {X 0,Y 428.533,Z 830.988,A -85,B 0,C 180,E1 20952.204,E2 20952.204} C_VEL
LIN {X 0,Y 430.378,Z 820.421,A -85,B 0,C 180,E1 20949.749,E2 20949.749} C_VEL
LIN {X 0,Y 432.559,Z 808.452,A -85,B 0,C 180,E1 20947.438,E2 20947.438} C_VEL
LIN {X 0,Y 434.998,Z 795.048,A -85,B 0,C 180,E1 20945.273,E2 20945.273} C_VEL
LIN {X 0,Y 437.67,Z 780.077,A -85,B 0,C 180,E1 20943.256,E2 20943.256} C_VEL
LIN {X 0,Y 440.327,Z 763.853,A -85,B 0,C 180,E1 20941.443,E2 20941.443} C_VEL
LIN {X 0,Y 442.774,Z 747.411,A -85,B 0,C 180,E1 20939.916,E2 20939.916} C_VEL
LIN {X 0,Y 445.166,Z 729.221,A -85,B 0,C 180,E1 20938.523,E2 20938.523} C_VEL
LIN {X 0,Y 447.177,Z 711.073,A -85,B 0,C 180,E1 20937.397,E2 20937.397} C_VEL
LIN {X 0,Y 448.827,Z 692.117,A -85,B 0,C 180,E1 20936.466,E2 20936.466} C_VEL
LIN {X 0,Y 450.058,Z 672.011,A -85,B 0,C 180,E1 20935.735,E2 20935.735} C_VEL
LIN {X 0,Y 450.776,Z 651.981,A -85,B 0,C 180,E1 20935.235,E2 20935.235} C_VEL
LIN {X 0,Y 455.755,Z 429.336,A -85,B 0,C 180,E1 20931.53,E2 20931.53} C_VEL
LIN {X 0,Y 443.658,Z 410.067,A -85,B 0,C 180,E1 20929.718,E2 20929.718} C_VEL
LIN {X 0,Y 432.706,Z 393.832,A -85,B 0,C 180,E1 20927.929,E2 20927.929} C_VEL
LIN {X 0,Y 427.135,Z 381.925,A -85,B 0,C 180,E1 20925.558,E2 20925.558} C_VEL
LIN {X 0,Y 425.422,Z 378.458,A -85,B 0,C 180,E1 20924.81,E2 20924.81} C_VEL
LIN {X 0,Y 425.311,Z 377.728,A -85,B 0,C 180,E1 20924.473,E2 20924.473} C_VEL
LIN {X 0,Y 425.298,Z 377.737,A -85,B 0,C 180,E1 20920.634,E2 20920.634} C_VEL
LIN {X 0,Y 425.284,Z 377.737,A -85,B 0,C 180,E1 20916.835,E2 20916.835} C_VEL
LIN {X 0,Y 425.284,Z 377.758,A -85,B 0,C 180,E1 20912.94,E2 20912.94} C_VEL
LIN {X 0,Y 425.291,Z 377.761,A -85,B 0,C 180,E1 20909.121,E2 20909.121} C_VEL
LIN {X 0,Y 425.306,Z 377.757,A -85,B 0,C 180,E1 20905.333,E2 20905.333} C_VEL
LIN {X 0,Y 425.326,Z 377.751,A -85,B 0,C 180,E1 20901.514,E2 20901.514} C_VEL
LIN {X 0,Y 425.306,Z 377.751,A -85,B 0,C 180,E1 20897.654,E2 20897.654} C_VEL
LIN {X 0,Y 425.272,Z 377.751,A -85,B 0,C 180,E1 20894.015,E2 20894.015} C_VEL
LIN {X 0,Y 425.263,Z 377.745,A -85,B 0,C 180,E1 20890.294,E2 20890.294} C_VEL
LIN {X 0,Y 425.277,Z 377.743,A -85,B 0,C 180,E1 20886.616,E2 20886.616} C_VEL
LIN {X 0,Y 425.297,Z 377.749,A -85,B 0,C 180,E1 20882.83,E2 20882.83} C_VEL
LIN {X 0,Y 425.299,Z 377.76,A -85,B 0,C 180,E1 20879.057,E2 20879.057} C_VEL
LIN {X 0,Y 425.266,Z 377.761,A -85,B 0,C 180,E1 20875.28,E2 20875.28} C_VEL
LIN {X 0,Y 425.246,Z 377.761,A -85,B 0,C 180,E1 20871.618,E2 20871.618} C_VEL
LIN {X 0,Y 425.245,Z 377.758,A -85,B 0,C 180,E1 20867.783,E2 20867.783} C_VEL
LIN {X 0,Y 425.272,Z 377.751,A -85,B 0,C 180,E1 20864.174,E2 20864.174} C_VEL
LIN {X 0,Y 425.29,Z 377.749,A -85,B 0,C 180,E1 20860.355,E2 20860.355} C_VEL
LIN {X 0,Y 425.255,Z 377.716,A -85,B 0,C 180,E1 20856.734,E2 20856.734} C_VEL
LIN {X 0,Y 425.247,Z 377.766,A -85,B 0,C 180,E1 20853.004,E2 20853.004} C_VEL
LIN {X 0,Y 425.245,Z 377.717,A -85,B 0,C 180,E1 20849.107,E2 20849.107} C_VEL
LIN {X 0,Y 425.263,Z 377.726,A -85,B 0,C 180,E1 20845.369,E2 20845.369} C_VEL
LIN {X 0,Y 425.298,Z 378.058,A -85,B 0,C 180,E1 20844.891,E2 20844.891} C_VEL
LIN {X 0,Y 426.57,Z 381.188,A -85,B 0,C 180,E1 20844.293,E2 20844.293} C_VEL
LIN {X 0,Y 427.841,Z 382.898,A -85,B 0,C 180,E1 20843.92,E2 20843.92} C_VEL
LIN {X 0,Y 429.663,Z 386.608,A -85,B 0,C 180,E1 20843.269,E2 20843.269} C_VEL
LIN {X 0,Y 437.213,Z 400.953,A -85,B 0,C 180,E1 20840.822,E2 20840.822} C_VEL
LIN {X 0,Y 446.013,Z 419.101,A -85,B 0,C 180,E1 20838.084,E2 20838.084} C_VEL
LIN {X 0,Y 454.266,Z 438.192,A -85,B 0,C 180,E1 20835.557,E2 20835.557} C_VEL
LIN {X 0,Y 453.595,Z 447.164,A -85,B 0,C 180,E1 20834.945,E2 20834.945} C_VEL
LIN {X 0,Y 458.012,Z 486.672,A -85,B 0,C 180,E1 20833.626,E2 20833.626} C_VEL
LIN {X 0,Y 451.636,Z 710.252,A -85,B 0,C 180,E1 20829.621,E2 20829.621} C_VEL
LIN {X 0,Y 450.275,Z 753.171,A -85,B 0,C 180,E1 20828.816,E2 20828.816} C_VEL
LIN {X 0,Y 448.67,Z 775.673,A -85,B 0,C 180,E1 20828.191,E2 20828.191} C_VEL
LIN {X 0,Y 446.765,Z 796.947,A -85,B 0,C 180,E1 20827.372,E2 20827.372} C_VEL
LIN {X 0,Y 444.62,Z 818.028,A -85,B 0,C 180,E1 20826.335,E2 20826.335} C_VEL
LIN {X 0,Y 442.189,Z 839.103,A -85,B 0,C 180,E1 20825.05,E2 20825.05} C_VEL
LIN {X 0,Y 439.653,Z 859.353,A -85,B 0,C 180,E1 20823.544,E2 20823.544} C_VEL
LIN {X 0,Y 437.025,Z 879.788,A -85,B 0,C 180,E1 20821.747,E2 20821.747} C_VEL
LIN {X 0,Y 434.684,Z 898.031,A -85,B 0,C 180,E1 20819.869,E2 20819.869} C_VEL
LIN {X 0,Y 432.386,Z 915.455,A -85,B 0,C 180,E1 20817.769,E2 20817.769} C_VEL
LIN {X 0,Y 430.391,Z 930.886,A -85,B 0,C 180,E1 20815.599,E2 20815.599} C_VEL
LIN {X 0,Y 428.606,Z 945.638,A -85,B 0,C 180,E1 20813.202,E2 20813.202} C_VEL
LIN {X 0,Y 427.127,Z 958.753,A -85,B 0,C 180,E1 20810.698,E2 20810.698} C_VEL
LIN {X 0,Y 425.942,Z 970.442,A -85,B 0,C 180,E1 20808.049,E2 20808.049} C_VEL
LIN {X 0,Y 425.062,Z 980.723,A -85,B 0,C 180,E1 20805.274,E2 20805.274} C_VEL
LIN {X 0,Y 424.505,Z 988.672,A -85,B 0,C 180,E1 20802.652,E2 20802.652} C_VEL
LIN {X 0,Y 424.144,Z 995.258,A -85,B 0,C 180,E1 20799.909,E2 20799.909} C_VEL
LIN {X 0,Y 423.969,Z 1000.02,A -85,B 0,C 180,E1 20797.316,E2 20797.316} C_VEL
LIN {X 0,Y 423.917,Z 1003.323,A -85,B 0,C 180,E1 20794.6,E2 20794.6} C_VEL
LIN {X 0,Y 423.903,Z 1005.117,A -85,B 0,C 180,E1 20791.893,E2 20791.893} C_VEL
LIN {X 0,Y 423.897,Z 1005.344,A -85,B 0,C 180,E1 20789.19,E2 20789.19} C_VEL
LIN {X 0,Y 423.912,Z 1004.261,A -85,B 0,C 180,E1 20786.485,E2 20786.485} C_VEL
LIN {X 0,Y 423.952,Z 1001.519,A -85,B 0,C 180,E1 20783.773,E2 20783.773} C_VEL
LIN {X 0,Y 424.074,Z 997.23,A -85,B 0,C 180,E1 20781.049,E2 20781.049} C_VEL
LIN {X 0,Y 424.35,Z 991.507,A -85,B 0,C 180,E1 20778.448,E2 20778.448} C_VEL
LIN {X 0,Y 424.813,Z 983.861,A -85,B 0,C 180,E1 20775.694,E2 20775.694} C_VEL
LIN {X 0,Y 425.547,Z 974.822,A -85,B 0,C 180,E1 20773.064,E2 20773.064} C_VEL
LIN {X 0,Y 426.578,Z 963.913,A -85,B 0,C 180,E1 20770.419,E2 20770.419} C_VEL
LIN {X 0,Y 427.899,Z 951.74,A -85,B 0,C 180,E1 20767.904,E2 20767.904} C_VEL
LIN {X 0,Y 429.515,Z 938.092,A -85,B 0,C 180,E1 20765.524,E2 20765.524} C_VEL
LIN {X 0,Y 431.516,Z 922.148,A -85,B 0,C 180,E1 20763.135,E2 20763.135} C_VEL
